KUKA KRL program: EPS_2_251806_MH06A_A_20260223023031.src

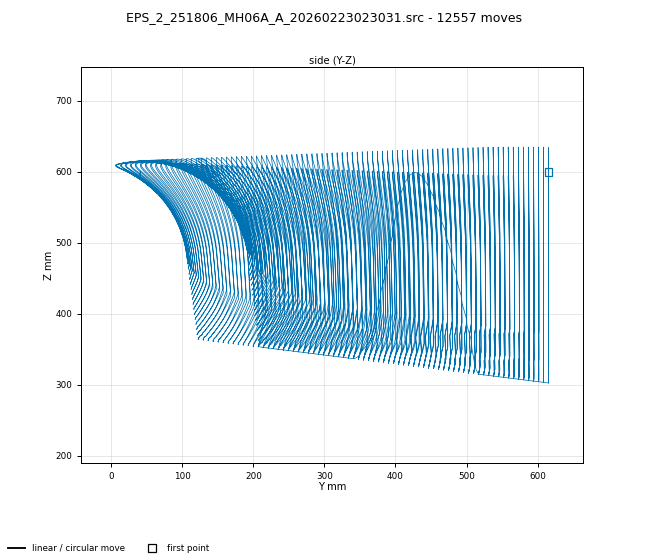
[picture p0: tool path of EPS_2_251806_MH06A_A_20260223023031.src, 12557 of 12559 moves have a stored position in this frame; points joined in program order, loops and branches not executed]
&ACCESS RVP
&REL 4
&COMMENT QRS 19112012
&PARAM EDITMASK = *
DEF PART()
EXT BAS (BAS_COMMAND :IN,REAL :IN )
INT I
BAS (#INITMOV,0 )

;KUKA QRS Post kuka4.cps  Date:22-06-2017 !

File_ID=3074

QRS_PRE_INIT()

;Init var - Until changes are made in qrs_pre_init
Outlet_Square_prg=0
Inlet_1_Square_prg=0
Inlet_2_Square_prg=0
Inlet_3_Square_prg=0
Inlet_4_Square_prg=0
Inlet_5_Square_prg=0

Outlet_1={X 0.000, Y 527.380, Z 509.000, B 0.000, E1 0.000 }
Inlet_1={X 0.000, Y 530.260, Z 469.000, B 0.000, E1 162.000 }
Outlet_1_type=251
Inlet_1_type=251
;QRS#1=Sidecore dimensions
;QRS#2=250-10" PVC SDR 35
;QRS#3=250-10" PVC SDR 35
;QRS#4=
;QRS#5=
;QRS#6=
;QRS#7=
;QRS#8=
;QRS#9=14M PSX
;QRS#10=14M PSX
;QRS#11=
;QRS#12=
;QRS#13=
;QRS#14=
;QRS#15=
;QRS#16=1220x127x914 3'
;QRS#17=EPS Height
;QRS#18=634,5
;QRS#19=*
;QRS#20= UPDATED VERSION 22-06-2017
;QRS#21=*
Outlet_Square=0100
Inlet_1_Square=0100
Inlet_2_Square=0
Inlet_3_Square=0
Inlet_4_Square=0
Inlet_5_Square=0
Mill_Square=1
Outlet_Square_Prg=205
Inlet_1_Square_prg=205

QRS_INIT()

$ADVANCE=5

; T1
PTP {E1 173.655,E2 173.655}
PTP {X 0,Y 615.421,A -85,B 0,C 180,E1 173.655,E2 173.655,E3 0,E4 0,E5 0,E6 0}
QRS_SPEED_INIT()
LIN {X 0,Y 615.421,Z 600,A -85,B 0,C 180,E1 173.655,E2 173.655,E3 0,E4 0,E5 0,E6 0} C_VEL
LIN {X 0,Y 615.421,Z 312.502,A -85,B 0,C 180,E1 173.655,E2 173.655} C_VEL
LIN {X 0,Y 615.421,Z 304.323,A -85,B 0,C 180,E1 173.655,E2 173.655} C_VEL
LIN {X 0,Y 615.418,Z 302.323,A -85,B 0,C 180,E1 173.469,E2 173.469} C_VEL
LIN {X 0,Y 615.458,Z 302.323,A -85,B 0,C 180,E1 170.801,E2 170.801} C_VEL
LIN {X 0,Y 615.445,Z 302.325,A -85,B 0,C 180,E1 168.139,E2 168.139} C_VEL
LIN {X 0,Y 615.434,Z 302.325,A -85,B 0,C 180,E1 166.083,E2 166.083} C_VEL
LIN {X 0,Y 615.411,Z 302.325,A -85,B 0,C 180,E1 163.589,E2 163.589} C_VEL
LIN {X 0,Y 615.423,Z 302.324,A -85,B 0,C 180,E1 161.352,E2 161.352} C_VEL
LIN {X 0,Y 615.489,Z 302.322,A -85,B 0,C 180,E1 158.568,E2 158.568} C_VEL
LIN {X 0,Y 615.423,Z 302.322,A -85,B 0,C 180,E1 155.726,E2 155.726} C_VEL
LIN {X 0,Y 615.484,Z 302.325,A -85,B 0,C 180,E1 152.953,E2 152.953} C_VEL
LIN {X 0,Y 615.446,Z 302.319,A -85,B 0,C 180,E1 150.21,E2 150.21} C_VEL
LIN {X 0,Y 615.435,Z 302.321,A -85,B 0,C 180,E1 147.675,E2 147.675} C_VEL
LIN {X 0,Y 615.476,Z 302.324,A -85,B 0,C 180,E1 145.185,E2 145.185} C_VEL
LIN {X 0,Y 615.492,Z 302.317,A -85,B 0,C 180,E1 142.759,E2 142.759} C_VEL
LIN {X 0,Y 615.452,Z 302.316,A -85,B 0,C 180,E1 140.247,E2 140.247} C_VEL
LIN {X 0,Y 615.453,Z 302.321,A -85,B 0,C 180,E1 137.645,E2 137.645} C_VEL
LIN {X 0,Y 615.489,Z 302.317,A -85,B 0,C 180,E1 134.932,E2 134.932} C_VEL
LIN {X 0,Y 615.456,Z 302.315,A -85,B 0,C 180,E1 132.354,E2 132.354} C_VEL
LIN {X 0,Y 615.46,Z 302.321,A -85,B 0,C 180,E1 129.751,E2 129.751} C_VEL
LIN {X 0,Y 615.455,Z 302.33,A -85,B 0,C 180,E1 128.039,E2 128.039} C_VEL
LIN {X 0,Y 615.471,Z 320.019,A -85,B 0,C 180,E1 125.415,E2 125.415} C_VEL
LIN {X 0,Y 615.484,Z 332.842,A -85,B 0,C 180,E1 123.534,E2 123.534} C_VEL
LIN {X 0,Y 615.493,Z 469.157,A -85,B 0,C 180,E1 121.905,E2 121.905} C_VEL
LIN {X 0,Y 615.496,Z 483.195,A -85,B 0,C 180,E1 121.609,E2 121.609} C_VEL
LIN {X 0,Y 615.493,Z 497.538,A -85,B 0,C 180,E1 121.162,E2 121.162} C_VEL
LIN {X 0,Y 615.494,Z 510.249,A -85,B 0,C 180,E1 120.633,E2 120.633} C_VEL
LIN {X 0,Y 615.49,Z 522.679,A -85,B 0,C 180,E1 119.978,E2 119.978} C_VEL
LIN {X 0,Y 615.497,Z 534.378,A -85,B 0,C 180,E1 119.217,E2 119.217} C_VEL
LIN {X 0,Y 615.498,Z 545.719,A -85,B 0,C 180,E1 118.318,E2 118.318} C_VEL
LIN {X 0,Y 615.496,Z 555.694,A -85,B 0,C 180,E1 117.36,E2 117.36} C_VEL
LIN {X 0,Y 615.495,Z 565.103,A -85,B 0,C 180,E1 116.26,E2 116.26} C_VEL
LIN {X 0,Y 615.495,Z 572.038,A -85,B 0,C 180,E1 115.281,E2 115.281} C_VEL
LIN {X 0,Y 615.495,Z 579.304,A -85,B 0,C 180,E1 114.011,E2 114.011} C_VEL
LIN {X 0,Y 615.493,Z 584.548,A -85,B 0,C 180,E1 112.843,E2 112.843} C_VEL
LIN {X 0,Y 615.498,Z 588.224,A -85,B 0,C 180,E1 111.783,E2 111.783} C_VEL
LIN {X 0,Y 615.493,Z 591.282,A -85,B 0,C 180,E1 110.559,E2 110.559} C_VEL
LIN {X 0,Y 615.491,Z 593.141,A -85,B 0,C 180,E1 109.337,E2 109.337} C_VEL
LIN {X 0,Y 615.498,Z 593.888,A -85,B 0,C 180,E1 107.956,E2 107.956} C_VEL
LIN {X 0,Y 615.489,Z 593.157,A -85,B 0,C 180,E1 106.586,E2 106.586} C_VEL
LIN {X 0,Y 615.493,Z 591.009,A -85,B 0,C 180,E1 105.225,E2 105.225} C_VEL
LIN {X 0,Y 615.499,Z 587.409,A -85,B 0,C 180,E1 103.873,E2 103.873} C_VEL
LIN {X 0,Y 615.491,Z 582.289,A -85,B 0,C 180,E1 102.529,E2 102.529} C_VEL
LIN {X 0,Y 615.496,Z 577.325,A -85,B 0,C 180,E1 101.526,E2 101.526} C_VEL
LIN {X 0,Y 615.496,Z 570.217,A -85,B 0,C 180,E1 100.36,E2 100.36} C_VEL
LIN {X 0,Y 615.496,Z 561.453,A -85,B 0,C 180,E1 99.198,E2 99.198} C_VEL
LIN {X 0,Y 615.497,Z 552.328,A -85,B 0,C 180,E1 98.205,E2 98.205} C_VEL
LIN {X 0,Y 615.496,Z 542.286,A -85,B 0,C 180,E1 97.297,E2 97.297} C_VEL
LIN {X 0,Y 615.5,Z 531.281,A -85,B 0,C 180,E1 96.474,E2 96.474} C_VEL
LIN {X 0,Y 615.489,Z 519.214,A -85,B 0,C 180,E1 95.733,E2 95.733} C_VEL
LIN {X 0,Y 615.495,Z 507.699,A -85,B 0,C 180,E1 95.158,E2 95.158} C_VEL
LIN {X 0,Y 615.496,Z 494.032,A -85,B 0,C 180,E1 94.625,E2 94.625} C_VEL
LIN {X 0,Y 615.492,Z 481.391,A -85,B 0,C 180,E1 94.256,E2 94.256} C_VEL
LIN {X 0,Y 615.492,Z 468.115,A -85,B 0,C 180,E1 93.989,E2 93.989} C_VEL
LIN {X 0,Y 615.476,Z 332.816,A -85,B 0,C 180,E1 92.372,E2 92.372} C_VEL
LIN {X 0,Y 615.478,Z 314.441,A -85,B 0,C 180,E1 89.672,E2 89.672} C_VEL
LIN {X 0,Y 615.448,Z 302.319,A -85,B 0,C 180,E1 87.852,E2 87.852} C_VEL
LIN {X 0,Y 615.458,Z 302.315,A -85,B 0,C 180,E1 85.415,E2 85.415} C_VEL
LIN {X 0,Y 615.494,Z 302.32,A -85,B 0,C 180,E1 82.784,E2 82.784} C_VEL
LIN {X 0,Y 615.448,Z 302.321,A -85,B 0,C 180,E1 80.137,E2 80.137} C_VEL
LIN {X 0,Y 615.445,Z 302.321,A -85,B 0,C 180,E1 78.138,E2 78.138} C_VEL
LIN {X 0,Y 615.441,Z 302.321,A -85,B 0,C 180,E1 76.084,E2 76.084} C_VEL
LIN {X 0,Y 615.447,Z 302.317,A -85,B 0,C 180,E1 73.581,E2 73.581} C_VEL
LIN {X 0,Y 615.477,Z 302.324,A -85,B 0,C 180,E1 70.661,E2 70.661} C_VEL
LIN {X 0,Y 615.458,Z 302.325,A -85,B 0,C 180,E1 68.567,E2 68.567} C_VEL
LIN {X 0,Y 615.429,Z 302.321,A -85,B 0,C 180,E1 66.003,E2 66.003} C_VEL
LIN {X 0,Y 615.448,Z 302.32,A -85,B 0,C 180,E1 63.554,E2 63.554} C_VEL
LIN {X 0,Y 615.448,Z 302.324,A -85,B 0,C 180,E1 60.591,E2 60.591} C_VEL
LIN {X 0,Y 615.426,Z 302.323,A -85,B 0,C 180,E1 58.311,E2 58.311} C_VEL
LIN {X 0,Y 615.422,Z 302.323,A -85,B 0,C 180,E1 55.974,E2 55.974} C_VEL
LIN {X 0,Y 615.449,Z 302.322,A -85,B 0,C 180,E1 53.572,E2 53.572} C_VEL
LIN {X 0,Y 615.467,Z 302.325,A -85,B 0,C 180,E1 50.94,E2 50.94} C_VEL
LIN {X 0,Y 615.421,Z 302.325,A -85,B 0,C 180,E1 48.52,E2 48.52} C_VEL
LIN {X 0,Y 615.424,Z 302.325,A -85,B 0,C 180,E1 45.844,E2 45.844} C_VEL
LIN {X 0,Y 615.466,Z 302.324,A -85,B 0,C 180,E1 43.045,E2 43.045} C_VEL
LIN {X 0,Y 615.422,Z 302.324,A -85,B 0,C 180,E1 40.611,E2 40.611} C_VEL
LIN {X 0,Y 615.426,Z 302.324,A -85,B 0,C 180,E1 38.004,E2 38.004} C_VEL
LIN {X 0,Y 615.469,Z 302.325,A -85,B 0,C 180,E1 35.617,E2 35.617} C_VEL
LIN {X 0,Y 615.483,Z 302.321,A -85,B 0,C 180,E1 33.236,E2 33.236} C_VEL
LIN {X 0,Y 615.447,Z 302.32,A -85,B 0,C 180,E1 30.922,E2 30.922} C_VEL
LIN {X 0,Y 615.426,Z 302.322,A -85,B 0,C 180,E1 28.439,E2 28.439} C_VEL
LIN {X 0,Y 615.476,Z 302.325,A -85,B 0,C 180,E1 25.716,E2 25.716} C_VEL
LIN {X 0,Y 615.438,Z 302.32,A -85,B 0,C 180,E1 22.846,E2 22.846} C_VEL
LIN {X 0,Y 615.433,Z 302.32,A -85,B 0,C 180,E1 20.543,E2 20.543} C_VEL
LIN {X 0,Y 615.467,Z 302.324,A -85,B 0,C 180,E1 17.957,E2 17.957} C_VEL
LIN {X 0,Y 615.475,Z 302.315,A -85,B 0,C 180,E1 15.226,E2 15.226} C_VEL
LIN {X 0,Y 615.44,Z 302.32,A -85,B 0,C 180,E1 12.531,E2 12.531} C_VEL
LIN {X 0,Y 615.497,Z 302.325,A -85,B 0,C 180,E1 9.862,E2 9.862} C_VEL
LIN {X 0,Y 615.47,Z 302.314,A -85,B 0,C 180,E1 7.216,E2 7.216} C_VEL
LIN {X 0,Y 615.473,Z 302.313,A -85,B 0,C 180,E1 5.241,E2 5.241} C_VEL
LIN {X 0,Y 615.447,Z 302.319,A -85,B 0,C 180,E1 2.618,E2 2.618} C_VEL
LIN {X 0,Y 615.487,Z 302.328,A -85,B 0,C 180,E1 0,E2 0} C_VEL
LIN {X 0,Y 615.484,Z 302.31,A -85,B 0,C 180,E1 -2.618,E2 -2.618} C_VEL
LIN {X 0,Y 615.454,Z 302.318,A -85,B 0,C 180,E1 -5.242,E2 -5.242} C_VEL
LIN {X 0,Y 615.487,Z 302.328,A -85,B 0,C 180,E1 -7.876,E2 -7.876} C_VEL
LIN {X 0,Y 615.49,Z 302.309,A -85,B 0,C 180,E1 -10.527,E2 -10.527} C_VEL
LIN {X 0,Y 615.46,Z 302.318,A -85,B 0,C 180,E1 -13.202,E2 -13.202} C_VEL
LIN {X 0,Y 615.491,Z 302.321,A -85,B 0,C 180,E1 -15.905,E2 -15.905} C_VEL
LIN {X 0,Y 615.477,Z 302.31,A -85,B 0,C 180,E1 -18.647,E2 -18.647} C_VEL
LIN {X 0,Y 615.481,Z 302.322,A -85,B 0,C 180,E1 -21.432,E2 -21.432} C_VEL
LIN {X 0,Y 615.491,Z 302.309,A -85,B 0,C 180,E1 -24.272,E2 -24.272} C_VEL
LIN {X 0,Y 615.469,Z 302.317,A -85,B 0,C 180,E1 -27.041,E2 -27.041} C_VEL
LIN {X 0,Y 615.482,Z 302.319,A -85,B 0,C 180,E1 -29.793,E2 -29.793} C_VEL
LIN {X 0,Y 615.488,Z 302.307,A -85,B 0,C 180,E1 -32.458,E2 -32.458} C_VEL
LIN {X 0,Y 615.473,Z 302.314,A -85,B 0,C 180,E1 -34.816,E2 -34.816} C_VEL
LIN {X 0,Y 615.484,Z 302.324,A -85,B 0,C 180,E1 -37.243,E2 -37.243} C_VEL
LIN {X 0,Y 615.487,Z 302.309,A -85,B 0,C 180,E1 -40.089,E2 -40.089} C_VEL
LIN {X 0,Y 615.493,Z 302.306,A -85,B 0,C 180,E1 -42.353,E2 -42.353} C_VEL
LIN {X 0,Y 615.48,Z 302.323,A -85,B 0,C 180,E1 -45.069,E2 -45.069} C_VEL
LIN {X 0,Y 615.479,Z 302.311,A -85,B 0,C 180,E1 -47.921,E2 -47.921} C_VEL
LIN {X 0,Y 615.494,Z 302.306,A -85,B 0,C 180,E1 -50.25,E2 -50.25} C_VEL
LIN {X 0,Y 615.485,Z 302.327,A -85,B 0,C 180,E1 -53.064,E2 -53.064} C_VEL
LIN {X 0,Y 615.481,Z 302.321,A -85,B 0,C 180,E1 -55.3,E2 -55.3} C_VEL
LIN {X 0,Y 615.468,Z 302.314,A -85,B 0,C 180,E1 -57.672,E2 -57.672} C_VEL
LIN {X 0,Y 615.497,Z 302.306,A -85,B 0,C 180,E1 -60.204,E2 -60.204} C_VEL
LIN {X 0,Y 615.498,Z 302.325,A -85,B 0,C 180,E1 -62.953,E2 -62.953} C_VEL
LIN {X 0,Y 615.469,Z 302.312,A -85,B 0,C 180,E1 -65.727,E2 -65.727} C_VEL
LIN {X 0,Y 615.483,Z 302.338,A -85,B 0,C 180,E1 -66.106,E2 -66.106} C_VEL
LIN {X 0,Y 615.484,Z 325.342,A -85,B 0,C 180,E1 -68.919,E2 -68.919} C_VEL
LIN {X 0,Y 615.5,Z 348.671,A -85,B 0,C 180,E1 -71.719,E2 -71.719} C_VEL
LIN {X 0,Y 615.483,Z 371.267,A -85,B 0,C 180,E1 -74.392,E2 -74.392} C_VEL
LIN {X 0,Y 615.498,Z 509.937,A -85,B 0,C 180,E1 -76.064,E2 -76.064} C_VEL
LIN {X 0,Y 615.495,Z 524.359,A -85,B 0,C 180,E1 -76.378,E2 -76.378} C_VEL
LIN {X 0,Y 615.489,Z 537.675,A -85,B 0,C 180,E1 -76.798,E2 -76.798} C_VEL
LIN {X 0,Y 615.498,Z 551.571,A -85,B 0,C 180,E1 -77.386,E2 -77.386} C_VEL
LIN {X 0,Y 615.495,Z 563.999,A -85,B 0,C 180,E1 -78.055,E2 -78.055} C_VEL
LIN {X 0,Y 615.499,Z 575.333,A -85,B 0,C 180,E1 -78.807,E2 -78.807} C_VEL
LIN {X 0,Y 615.498,Z 585.742,A -85,B 0,C 180,E1 -79.639,E2 -79.639} C_VEL
LIN {X 0,Y 615.496,Z 596.083,A -85,B 0,C 180,E1 -80.635,E2 -80.635} C_VEL
LIN {X 0,Y 615.497,Z 604.598,A -85,B 0,C 180,E1 -81.628,E2 -81.628} C_VEL
LIN {X 0,Y 615.496,Z 612.723,A -85,B 0,C 180,E1 -82.784,E2 -82.784} C_VEL
LIN {X 0,Y 615.496,Z 618.427,A -85,B 0,C 180,E1 -83.772,E2 -83.772} C_VEL
LIN {X 0,Y 615.495,Z 623.078,A -85,B 0,C 180,E1 -84.758,E2 -84.758} C_VEL
LIN {X 0,Y 615.494,Z 627.9,A -85,B 0,C 180,E1 -86.071,E2 -86.071} C_VEL
LIN {X 0,Y 615.496,Z 631.251,A -85,B 0,C 180,E1 -87.382,E2 -87.382} C_VEL
LIN {X 0,Y 615.489,Z 633.228,A -85,B 0,C 180,E1 -88.691,E2 -88.691} C_VEL
LIN {X 0,Y 615.493,Z 633.889,A -85,B 0,C 180,E1 -89.999,E2 -89.999} C_VEL
LIN {X 0,Y 615.489,Z 633.229,A -85,B 0,C 180,E1 -91.308,E2 -91.308} C_VEL
LIN {X 0,Y 615.496,Z 631.253,A -85,B 0,C 180,E1 -92.617,E2 -92.617} C_VEL
LIN {X 0,Y 615.494,Z 627.904,A -85,B 0,C 180,E1 -93.928,E2 -93.928} C_VEL
LIN {X 0,Y 615.495,Z 623.083,A -85,B 0,C 180,E1 -95.24,E2 -95.24} C_VEL
LIN {X 0,Y 615.496,Z 616.632,A -85,B 0,C 180,E1 -96.556,E2 -96.556} C_VEL
LIN {X 0,Y 615.497,Z 609.445,A -85,B 0,C 180,E1 -97.71,E2 -97.71} C_VEL
LIN {X 0,Y 615.497,Z 601.908,A -85,B 0,C 180,E1 -98.701,E2 -98.701} C_VEL
LIN {X 0,Y 615.495,Z 592.859,A -85,B 0,C 180,E1 -99.695,E2 -99.695} C_VEL
LIN {X 0,Y 615.497,Z 582.763,A -85,B 0,C 180,E1 -100.618,E2 -100.618} C_VEL
LIN {X 0,Y 615.498,Z 571.867,A -85,B 0,C 180,E1 -101.442,E2 -101.442} C_VEL
LIN {X 0,Y 615.489,Z 559.718,A -85,B 0,C 180,E1 -102.195,E2 -102.195} C_VEL
LIN {X 0,Y 615.498,Z 546.106,A -85,B 0,C 180,E1 -102.865,E2 -102.865} C_VEL
LIN {X 0,Y 615.49,Z 532.855,A -85,B 0,C 180,E1 -103.368,E2 -103.368} C_VEL
LIN {X 0,Y 615.494,Z 519.315,A -85,B 0,C 180,E1 -103.747,E2 -103.747} C_VEL
LIN {X 0,Y 615.493,Z 504.752,A -85,B 0,C 180,E1 -104.013,E2 -104.013} C_VEL
LIN {X 0,Y 615.483,Z 371.277,A -85,B 0,C 180,E1 -105.607,E2 -105.607} C_VEL
LIN {X 0,Y 615.49,Z 347.317,A -85,B 0,C 180,E1 -108.442,E2 -108.442} C_VEL
LIN {X 0,Y 615.486,Z 325.352,A -85,B 0,C 180,E1 -111.08,E2 -111.08} C_VEL
LIN {X 0,Y 615.484,Z 302.309,A -85,B 0,C 180,E1 -113.908,E2 -113.908} C_VEL
LIN {X 0,Y 615.466,Z 302.316,A -85,B 0,C 180,E1 -116.444,E2 -116.444} C_VEL
LIN {X 0,Y 615.474,Z 302.319,A -85,B 0,C 180,E1 -118.658,E2 -118.658} C_VEL
LIN {X 0,Y 615.485,Z 302.324,A -85,B 0,C 180,E1 -121.085,E2 -121.085} C_VEL
LIN {X 0,Y 615.482,Z 302.309,A -85,B 0,C 180,E1 -124.021,E2 -124.021} C_VEL
LIN {X 0,Y 615.476,Z 302.317,A -85,B 0,C 180,E1 -126.424,E2 -126.424} C_VEL
LIN {X 0,Y 615.482,Z 302.32,A -85,B 0,C 180,E1 -129.061,E2 -129.061} C_VEL
LIN {X 0,Y 615.48,Z 302.311,A -85,B 0,C 180,E1 -131.473,E2 -131.473} C_VEL
LIN {X 0,Y 615.481,Z 302.314,A -85,B 0,C 180,E1 -134.149,E2 -134.149} C_VEL
LIN {X 0,Y 615.477,Z 302.319,A -85,B 0,C 180,E1 -136.952,E2 -136.952} C_VEL
LIN {X 0,Y 615.475,Z 302.311,A -85,B 0,C 180,E1 -139.392,E2 -139.392} C_VEL
LIN {X 0,Y 615.487,Z 302.312,A -85,B 0,C 180,E1 -141.987,E2 -141.987} C_VEL
LIN {X 0,Y 615.495,Z 302.323,A -85,B 0,C 180,E1 -144.384,E2 -144.384} C_VEL
LIN {X 0,Y 615.471,Z 302.32,A -85,B 0,C 180,E1 -146.763,E2 -146.763} C_VEL
LIN {X 0,Y 615.462,Z 302.315,A -85,B 0,C 180,E1 -149.079,E2 -149.079} C_VEL
LIN {X 0,Y 615.488,Z 302.309,A -85,B 0,C 180,E1 -151.548,E2 -151.548} C_VEL
LIN {X 0,Y 615.481,Z 302.323,A -85,B 0,C 180,E1 -154.43,E2 -154.43} C_VEL
LIN {X 0,Y 615.459,Z 302.314,A -85,B 0,C 180,E1 -157.154,E2 -157.154} C_VEL
LIN {X 0,Y 615.493,Z 302.32,A -85,B 0,C 180,E1 -159.967,E2 -159.967} C_VEL
LIN {X 0,Y 615.447,Z 302.319,A -85,B 0,C 180,E1 -162.728,E2 -162.728} C_VEL
LIN {X 0,Y 615.484,Z 302.312,A -85,B 0,C 180,E1 -165.451,E2 -165.451} C_VEL
LIN {X 0,Y 615.479,Z 302.324,A -85,B 0,C 180,E1 -168.139,E2 -168.139} C_VEL
LIN {X 0,Y 615.44,Z 302.319,A -85,B 0,C 180,E1 -170.8,E2 -170.8} C_VEL
LIN {X 0,Y 615.487,Z 302.315,A -85,B 0,C 180,E1 -173.443,E2 -173.443} C_VEL
LIN {X 0,Y 615.465,Z 302.324,A -85,B 0,C 180,E1 -176.071,E2 -176.071} C_VEL
LIN {X 0,Y 615.429,Z 302.321,A -85,B 0,C 180,E1 -178.691,E2 -178.691} C_VEL
LIN {X 0,Y 615.473,Z 302.319,A -85,B 0,C 180,E1 -181.308,E2 -181.308} C_VEL
LIN {X 0,Y 615.46,Z 302.324,A -85,B 0,C 180,E1 -183.928,E2 -183.928} C_VEL
LIN {X 0,Y 615.418,Z 302.323,A -85,B 0,C 180,E1 -186.531,E2 -186.531} C_VEL
LIN {X 0,Y 614.771,Z 302.471,A -85,B 0,C 180,E1 -187.077,E2 -187.077} C_VEL
LIN {X 0,Y 611.962,Z 302.879,A -85,B 0,C 180,E1 -187.963,E2 -187.963} C_VEL
LIN {X 0,Y 609.571,Z 303.192,A -85,B 0,C 180,E1 -188.676,E2 -188.676} C_VEL
LIN {X 0,Y 608.527,Z 303.311,A -85,B 0,C 180,E1 -189.225,E2 -189.225} C_VEL
LIN {X 0,Y 608.433,Z 303.32,A -85,B 0,C 180,E1 -189.412,E2 -189.412} C_VEL
LIN {X 0,Y 608.418,Z 303.319,A -85,B 0,C 180,E1 -192,E2 -192} C_VEL
LIN {X 0,Y 608.406,Z 303.32,A -85,B 0,C 180,E1 -194.039,E2 -194.039} C_VEL
LIN {X 0,Y 608.384,Z 303.321,A -85,B 0,C 180,E1 -196.506,E2 -196.506} C_VEL
LIN {X 0,Y 608.425,Z 303.319,A -85,B 0,C 180,E1 -198.87,E2 -198.87} C_VEL
LIN {X 0,Y 608.447,Z 303.317,A -85,B 0,C 180,E1 -201.692,E2 -201.692} C_VEL
LIN {X 0,Y 608.416,Z 303.319,A -85,B 0,C 180,E1 -204.572,E2 -204.572} C_VEL
LIN {X 0,Y 608.477,Z 303.319,A -85,B 0,C 180,E1 -207.209,E2 -207.209} C_VEL
LIN {X 0,Y 608.409,Z 303.318,A -85,B 0,C 180,E1 -209.964,E2 -209.964} C_VEL
LIN {X 0,Y 608.422,Z 303.319,A -85,B 0,C 180,E1 -212.518,E2 -212.518} C_VEL
LIN {X 0,Y 608.425,Z 303.321,A -85,B 0,C 180,E1 -215.278,E2 -215.278} C_VEL
LIN {X 0,Y 608.442,Z 303.314,A -85,B 0,C 180,E1 -217.748,E2 -217.748} C_VEL
LIN {X 0,Y 608.422,Z 303.318,A -85,B 0,C 180,E1 -220.327,E2 -220.327} C_VEL
LIN {X 0,Y 608.455,Z 303.32,A -85,B 0,C 180,E1 -222.959,E2 -222.959} C_VEL
LIN {X 0,Y 608.425,Z 303.316,A -85,B 0,C 180,E1 -225.739,E2 -225.739} C_VEL
LIN {X 0,Y 608.43,Z 303.316,A -85,B 0,C 180,E1 -227.937,E2 -227.937} C_VEL
LIN {X 0,Y 608.471,Z 303.321,A -85,B 0,C 180,E1 -230.702,E2 -230.702} C_VEL
LIN {X 0,Y 608.45,Z 303.347,A -85,B 0,C 180,E1 -231.87,E2 -231.87} C_VEL
LIN {X 0,Y 608.5,Z 319.687,A -85,B 0,C 180,E1 -234.321,E2 -234.321} C_VEL
LIN {X 0,Y 608.532,Z 333.181,A -85,B 0,C 180,E1 -236.289,E2 -236.289} C_VEL
LIN {X 0,Y 608.603,Z 469.47,A -85,B 0,C 180,E1 -237.939,E2 -237.939} C_VEL
LIN {X 0,Y 608.596,Z 483.994,A -85,B 0,C 180,E1 -238.255,E2 -238.255} C_VEL
LIN {X 0,Y 608.56,Z 497.685,A -85,B 0,C 180,E1 -238.69,E2 -238.69} C_VEL
LIN {X 0,Y 608.538,Z 511.282,A -85,B 0,C 180,E1 -239.268,E2 -239.268} C_VEL
LIN {X 0,Y 608.529,Z 523.689,A -85,B 0,C 180,E1 -239.938,E2 -239.938} C_VEL
LIN {X 0,Y 608.518,Z 535.16,A -85,B 0,C 180,E1 -240.699,E2 -240.699} C_VEL
LIN {X 0,Y 608.503,Z 546.875,A -85,B 0,C 180,E1 -241.646,E2 -241.646} C_VEL
LIN {X 0,Y 608.476,Z 557.274,A -85,B 0,C 180,E1 -242.674,E2 -242.674} C_VEL
LIN {X 0,Y 608.465,Z 566.452,A -85,B 0,C 180,E1 -243.782,E2 -243.782} C_VEL
LIN {X 0,Y 608.454,Z 573.946,A -85,B 0,C 180,E1 -244.883,E2 -244.883} C_VEL
LIN {X 0,Y 608.444,Z 580.901,A -85,B 0,C 180,E1 -246.155,E2 -246.155} C_VEL
LIN {X 0,Y 608.422,Z 585.559,A -85,B 0,C 180,E1 -247.235,E2 -247.235} C_VEL
LIN {X 0,Y 608.427,Z 589.176,A -85,B 0,C 180,E1 -248.308,E2 -248.308} C_VEL
LIN {X 0,Y 608.435,Z 592.445,A -85,B 0,C 180,E1 -249.726,E2 -249.726} C_VEL
LIN {X 0,Y 608.424,Z 594.154,A -85,B 0,C 180,E1 -251.13,E2 -251.13} C_VEL
LIN {X 0,Y 608.415,Z 594.394,A -85,B 0,C 180,E1 -252.523,E2 -252.523} C_VEL
LIN {X 0,Y 608.431,Z 593.195,A -85,B 0,C 180,E1 -253.906,E2 -253.906} C_VEL
LIN {X 0,Y 608.42,Z 590.521,A -85,B 0,C 180,E1 -255.279,E2 -255.279} C_VEL
LIN {X 0,Y 608.441,Z 586.343,A -85,B 0,C 180,E1 -256.644,E2 -256.644} C_VEL
LIN {X 0,Y 608.444,Z 580.582,A -85,B 0,C 180,E1 -258.001,E2 -258.001} C_VEL
LIN {X 0,Y 608.435,Z 574.844,A -85,B 0,C 180,E1 -259.059,E2 -259.059} C_VEL
LIN {X 0,Y 608.45,Z 567.318,A -85,B 0,C 180,E1 -260.191,E2 -260.191} C_VEL
LIN {X 0,Y 608.475,Z 559.21,A -85,B 0,C 180,E1 -261.198,E2 -261.198} C_VEL
LIN {X 0,Y 608.492,Z 549.496,A -85,B 0,C 180,E1 -262.201,E2 -262.201} C_VEL
LIN {X 0,Y 608.511,Z 538.671,A -85,B 0,C 180,E1 -263.127,E2 -263.127} C_VEL
LIN {X 0,Y 608.532,Z 526.982,A -85,B 0,C 180,E1 -263.951,E2 -263.951} C_VEL
LIN {X 0,Y 608.532,Z 513.82,A -85,B 0,C 180,E1 -264.699,E2 -264.699} C_VEL
LIN {X 0,Y 608.575,Z 500.825,A -85,B 0,C 180,E1 -265.281,E2 -265.281} C_VEL
LIN {X 0,Y 608.589,Z 486.737,A -85,B 0,C 180,E1 -265.758,E2 -265.758} C_VEL
LIN {X 0,Y 608.604,Z 472.745,A -85,B 0,C 180,E1 -266.09,E2 -266.09} C_VEL
LIN {X 0,Y 608.618,Z 453.41,A -85,B 0,C 180,E1 -266.359,E2 -266.359} C_VEL
LIN {X 0,Y 608.493,Z 332.936,A -85,B 0,C 180,E1 -267.808,E2 -267.808} C_VEL
LIN {X 0,Y 608.514,Z 313.697,A -85,B 0,C 180,E1 -270.662,E2 -270.662} C_VEL
LIN {X 0,Y 608.434,Z 303.317,A -85,B 0,C 180,E1 -272.235,E2 -272.235} C_VEL
LIN {X 0,Y 608.43,Z 303.316,A -85,B 0,C 180,E1 -274.638,E2 -274.638} C_VEL
LIN {X 0,Y 608.484,Z 303.318,A -85,B 0,C 180,E1 -277.3,E2 -277.3} C_VEL
LIN {X 0,Y 608.421,Z 303.318,A -85,B 0,C 180,E1 -279.978,E2 -279.978} C_VEL
LIN {X 0,Y 608.428,Z 303.316,A -85,B 0,C 180,E1 -282.001,E2 -282.001} C_VEL
LIN {X 0,Y 608.417,Z 303.317,A -85,B 0,C 180,E1 -284.039,E2 -284.039} C_VEL
LIN {X 0,Y 608.445,Z 303.314,A -85,B 0,C 180,E1 -286.523,E2 -286.523} C_VEL
LIN {X 0,Y 608.43,Z 303.319,A -85,B 0,C 180,E1 -289.572,E2 -289.572} C_VEL
LIN {X 0,Y 608.431,Z 303.316,A -85,B 0,C 180,E1 -292.407,E2 -292.407} C_VEL
LIN {X 0,Y 608.429,Z 303.322,A -85,B 0,C 180,E1 -295.302,E2 -295.302} C_VEL
LIN {X 0,Y 608.423,Z 303.319,A -85,B 0,C 180,E1 -297.52,E2 -297.52} C_VEL
LIN {X 0,Y 608.395,Z 303.32,A -85,B 0,C 180,E1 -299.96,E2 -299.96} C_VEL
LIN {X 0,Y 608.432,Z 303.318,A -85,B 0,C 180,E1 -302.519,E2 -302.519} C_VEL
LIN {X 0,Y 608.414,Z 303.322,A -85,B 0,C 180,E1 -305.28,E2 -305.28} C_VEL
LIN {X 0,Y 608.396,Z 303.319,A -85,B 0,C 180,E1 -307.752,E2 -307.752} C_VEL
LIN {X 0,Y 608.432,Z 303.318,A -85,B 0,C 180,E1 -310.327,E2 -310.327} C_VEL
LIN {X 0,Y 608.428,Z 303.318,A -85,B 0,C 180,E1 -313.305,E2 -313.305} C_VEL
LIN {X 0,Y 608.418,Z 303.318,A -85,B 0,C 180,E1 -316.126,E2 -316.126} C_VEL
LIN {X 0,Y 608.439,Z 303.322,A -85,B 0,C 180,E1 -318.822,E2 -318.822} C_VEL
LIN {X 0,Y 608.396,Z 303.32,A -85,B 0,C 180,E1 -321.407,E2 -321.407} C_VEL
LIN {X 0,Y 608.424,Z 303.317,A -85,B 0,C 180,E1 -323.907,E2 -323.907} C_VEL
LIN {X 0,Y 608.443,Z 303.32,A -85,B 0,C 180,E1 -326.328,E2 -326.328} C_VEL
LIN {X 0,Y 608.44,Z 303.321,A -85,B 0,C 180,E1 -328.734,E2 -328.734} C_VEL
LIN {X 0,Y 608.424,Z 303.316,A -85,B 0,C 180,E1 -331.389,E2 -331.389} C_VEL
LIN {X 0,Y 608.416,Z 303.32,A -85,B 0,C 180,E1 -333.963,E2 -333.963} C_VEL
LIN {X 0,Y 608.426,Z 303.318,A -85,B 0,C 180,E1 -336.875,E2 -336.875} C_VEL
LIN {X 0,Y 608.427,Z 303.316,A -85,B 0,C 180,E1 -339.332,E2 -339.332} C_VEL
LIN {X 0,Y 608.419,Z 303.32,A -85,B 0,C 180,E1 -341.827,E2 -341.827} C_VEL
LIN {X 0,Y 608.46,Z 303.316,A -85,B 0,C 180,E1 -344.594,E2 -344.594} C_VEL
LIN {X 0,Y 608.415,Z 303.317,A -85,B 0,C 180,E1 -347.322,E2 -347.322} C_VEL
LIN {X 0,Y 608.457,Z 303.32,A -85,B 0,C 180,E1 -350.023,E2 -350.023} C_VEL
LIN {X 0,Y 608.439,Z 303.316,A -85,B 0,C 180,E1 -352.701,E2 -352.701} C_VEL
LIN {X 0,Y 608.455,Z 303.314,A -85,B 0,C 180,E1 -354.698,E2 -354.698} C_VEL
LIN {X 0,Y 608.443,Z 303.315,A -85,B 0,C 180,E1 -357.352,E2 -357.352} C_VEL
LIN {X 0,Y 608.477,Z 303.32,A -85,B 0,C 180,E1 -360,E2 -360} C_VEL
LIN {X 0,Y 608.474,Z 303.311,A -85,B 0,C 180,E1 -362.648,E2 -362.648} C_VEL
LIN {X 0,Y 608.439,Z 303.316,A -85,B 0,C 180,E1 -365.302,E2 -365.302} C_VEL
LIN {X 0,Y 608.478,Z 303.318,A -85,B 0,C 180,E1 -367.967,E2 -367.967} C_VEL
LIN {X 0,Y 608.458,Z 303.312,A -85,B 0,C 180,E1 -370.949,E2 -370.949} C_VEL
LIN {X 0,Y 608.447,Z 303.317,A -85,B 0,C 180,E1 -373.357,E2 -373.357} C_VEL
LIN {X 0,Y 608.465,Z 303.315,A -85,B 0,C 180,E1 -376.094,E2 -376.094} C_VEL
LIN {X 0,Y 608.45,Z 303.313,A -85,B 0,C 180,E1 -378.87,E2 -378.87} C_VEL
LIN {X 0,Y 608.465,Z 303.321,A -85,B 0,C 180,E1 -381.692,E2 -381.692} C_VEL
LIN {X 0,Y 608.449,Z 303.313,A -85,B 0,C 180,E1 -384.571,E2 -384.571} C_VEL
LIN {X 0,Y 608.469,Z 303.315,A -85,B 0,C 180,E1 -387.205,E2 -387.205} C_VEL
LIN {X 0,Y 608.466,Z 303.314,A -85,B 0,C 180,E1 -389.971,E2 -389.971} C_VEL
LIN {X 0,Y 608.458,Z 303.314,A -85,B 0,C 180,E1 -392.88,E2 -392.88} C_VEL
LIN {X 0,Y 608.439,Z 303.323,A -85,B 0,C 180,E1 -395.278,E2 -395.278} C_VEL
LIN {X 0,Y 608.468,Z 303.315,A -85,B 0,C 180,E1 -397.747,E2 -397.747} C_VEL
LIN {X 0,Y 608.449,Z 303.313,A -85,B 0,C 180,E1 -400.328,E2 -400.328} C_VEL
LIN {X 0,Y 608.483,Z 303.319,A -85,B 0,C 180,E1 -403.31,E2 -403.31} C_VEL
LIN {X 0,Y 608.468,Z 303.311,A -85,B 0,C 180,E1 -406.13,E2 -406.13} C_VEL
LIN {X 0,Y 608.453,Z 303.317,A -85,B 0,C 180,E1 -408.823,E2 -408.823} C_VEL
LIN {X 0,Y 608.471,Z 303.316,A -85,B 0,C 180,E1 -411.412,E2 -411.412} C_VEL
LIN {X 0,Y 608.449,Z 303.313,A -85,B 0,C 180,E1 -413.954,E2 -413.954} C_VEL
LIN {X 0,Y 608.451,Z 303.313,A -85,B 0,C 180,E1 -416.328,E2 -416.328} C_VEL
LIN {X 0,Y 608.45,Z 303.319,A -85,B 0,C 180,E1 -418.732,E2 -418.732} C_VEL
LIN {X 0,Y 608.46,Z 303.315,A -85,B 0,C 180,E1 -421.383,E2 -421.383} C_VEL
LIN {X 0,Y 608.44,Z 303.314,A -85,B 0,C 180,E1 -423.964,E2 -423.964} C_VEL
LIN {X 0,Y 608.484,Z 303.496,A -85,B 0,C 180,E1 -425.959,E2 -425.959} C_VEL
LIN {X 0,Y 608.598,Z 318.101,A -85,B 0,C 180,E1 -427.778,E2 -427.778} C_VEL
LIN {X 0,Y 608.579,Z 339.823,A -85,B 0,C 180,E1 -430.433,E2 -430.433} C_VEL
LIN {X 0,Y 608.526,Z 362.995,A -85,B 0,C 180,E1 -433.218,E2 -433.218} C_VEL
LIN {X 0,Y 608.51,Z 371.412,A -85,B 0,C 180,E1 -434.219,E2 -434.219} C_VEL
LIN {X 0,Y 608.617,Z 509.424,A -85,B 0,C 180,E1 -435.894,E2 -435.894} C_VEL
LIN {X 0,Y 608.594,Z 523.606,A -85,B 0,C 180,E1 -436.199,E2 -436.199} C_VEL
LIN {X 0,Y 608.579,Z 537.697,A -85,B 0,C 180,E1 -436.646,E2 -436.646} C_VEL
LIN {X 0,Y 608.565,Z 549.872,A -85,B 0,C 180,E1 -437.155,E2 -437.155} C_VEL
LIN {X 0,Y 608.516,Z 562.671,A -85,B 0,C 180,E1 -437.832,E2 -437.832} C_VEL
LIN {X 0,Y 608.499,Z 575.463,A -85,B 0,C 180,E1 -438.676,E2 -438.676} C_VEL
LIN {X 0,Y 608.496,Z 585.925,A -85,B 0,C 180,E1 -439.518,E2 -439.518} C_VEL
LIN {X 0,Y 608.479,Z 596.329,A -85,B 0,C 180,E1 -440.526,E2 -440.526} C_VEL
LIN {X 0,Y 608.464,Z 604.909,A -85,B 0,C 180,E1 -441.531,E2 -441.531} C_VEL
LIN {X 0,Y 608.461,Z 613.11,A -85,B 0,C 180,E1 -442.7,E2 -442.7} C_VEL
LIN {X 0,Y 608.443,Z 619.544,A -85,B 0,C 180,E1 -443.831,E2 -443.831} C_VEL
LIN {X 0,Y 608.438,Z 624.96,A -85,B 0,C 180,E1 -445.03,E2 -445.03} C_VEL
LIN {X 0,Y 608.432,Z 628.439,A -85,B 0,C 180,E1 -446.025,E2 -446.025} C_VEL
LIN {X 0,Y 608.424,Z 631.83,A -85,B 0,C 180,E1 -447.351,E2 -447.351} C_VEL
LIN {X 0,Y 608.442,Z 633.83,A -85,B 0,C 180,E1 -448.676,E2 -448.676} C_VEL
LIN {X 0,Y 608.433,Z 634.5,A -85,B 0,C 180,E1 -449.999,E2 -449.999} C_VEL
LIN {X 0,Y 608.442,Z 633.831,A -85,B 0,C 180,E1 -451.323,E2 -451.323} C_VEL
LIN {X 0,Y 608.424,Z 631.832,A -85,B 0,C 180,E1 -452.648,E2 -452.648} C_VEL
LIN {X 0,Y 608.431,Z 628.443,A -85,B 0,C 180,E1 -453.973,E2 -453.973} C_VEL
LIN {X 0,Y 608.44,Z 623.57,A -85,B 0,C 180,E1 -455.301,E2 -455.301} C_VEL
LIN {X 0,Y 608.445,Z 617.214,A -85,B 0,C 180,E1 -456.603,E2 -456.603} C_VEL
LIN {X 0,Y 608.453,Z 609.802,A -85,B 0,C 180,E1 -457.8,E2 -457.8} C_VEL
LIN {X 0,Y 608.472,Z 600.829,A -85,B 0,C 180,E1 -458.97,E2 -458.97} C_VEL
LIN {X 0,Y 608.472,Z 591.398,A -85,B 0,C 180,E1 -459.976,E2 -459.976} C_VEL
LIN {X 0,Y 608.505,Z 580.051,A -85,B 0,C 180,E1 -460.973,E2 -460.973} C_VEL
LIN {X 0,Y 608.533,Z 568.158,A -85,B 0,C 180,E1 -461.829,E2 -461.829} C_VEL
LIN {X 0,Y 608.531,Z 555.085,A -85,B 0,C 180,E1 -462.59,E2 -462.59} C_VEL
LIN {X 0,Y 608.556,Z 542.188,A -85,B 0,C 180,E1 -463.184,E2 -463.184} C_VEL
LIN {X 0,Y 608.593,Z 528.205,A -85,B 0,C 180,E1 -463.672,E2 -463.672} C_VEL
LIN {X 0,Y 608.62,Z 514.489,A -85,B 0,C 180,E1 -464.012,E2 -464.012} C_VEL
LIN {X 0,Y 608.62,Z 498.221,A -85,B 0,C 180,E1 -464.257,E2 -464.257} C_VEL
LIN {X 0,Y 608.524,Z 371.423,A -85,B 0,C 180,E1 -465.78,E2 -465.78} C_VEL
LIN {X 0,Y 608.563,Z 346.655,A -85,B 0,C 180,E1 -468.741,E2 -468.741} C_VEL
LIN {X 0,Y 608.588,Z 322.456,A -85,B 0,C 180,E1 -471.686,E2 -471.686} C_VEL
LIN {X 0,Y 608.541,Z 303.719,A -85,B 0,C 180,E1 -474.011,E2 -474.011} C_VEL
LIN {X 0,Y 608.461,Z 303.314,A -85,B 0,C 180,E1 -474.071,E2 -474.071} C_VEL
LIN {X 0,Y 608.445,Z 303.319,A -85,B 0,C 180,E1 -476.774,E2 -476.774} C_VEL
LIN {X 0,Y 608.481,Z 303.31,A -85,B 0,C 180,E1 -479.778,E2 -479.778} C_VEL
LIN {X 0,Y 608.448,Z 303.317,A -85,B 0,C 180,E1 -482.52,E2 -482.52} C_VEL
LIN {X 0,Y 608.447,Z 303.317,A -85,B 0,C 180,E1 -485.276,E2 -485.276} C_VEL
LIN {X 0,Y 608.466,Z 303.311,A -85,B 0,C 180,E1 -487.745,E2 -487.745} C_VEL
LIN {X 0,Y 608.447,Z 303.317,A -85,B 0,C 180,E1 -490.328,E2 -490.328} C_VEL
LIN {X 0,Y 608.445,Z 303.32,A -85,B 0,C 180,E1 -492.959,E2 -492.959} C_VEL
LIN {X 0,Y 608.459,Z 303.312,A -85,B 0,C 180,E1 -495.735,E2 -495.735} C_VEL
LIN {X 0,Y 608.463,Z 303.321,A -85,B 0,C 180,E1 -498.656,E2 -498.656} C_VEL
LIN {X 0,Y 608.459,Z 303.312,A -85,B 0,C 180,E1 -501.411,E2 -501.411} C_VEL
LIN {X 0,Y 608.474,Z 303.312,A -85,B 0,C 180,E1 -503.949,E2 -503.949} C_VEL
LIN {X 0,Y 608.469,Z 303.319,A -85,B 0,C 180,E1 -506.329,E2 -506.329} C_VEL
LIN {X 0,Y 608.437,Z 303.319,A -85,B 0,C 180,E1 -508.732,E2 -508.732} C_VEL
LIN {X 0,Y 608.466,Z 303.311,A -85,B 0,C 180,E1 -511.379,E2 -511.379} C_VEL
LIN {X 0,Y 608.474,Z 303.321,A -85,B 0,C 180,E1 -514.276,E2 -514.276} C_VEL
LIN {X 0,Y 608.432,Z 303.316,A -85,B 0,C 180,E1 -516.875,E2 -516.875} C_VEL
LIN {X 0,Y 608.463,Z 303.315,A -85,B 0,C 180,E1 -519.726,E2 -519.726} C_VEL
LIN {X 0,Y 608.431,Z 303.319,A -85,B 0,C 180,E1 -522.523,E2 -522.523} C_VEL
LIN {X 0,Y 608.463,Z 303.312,A -85,B 0,C 180,E1 -525.279,E2 -525.279} C_VEL
LIN {X 0,Y 608.454,Z 303.323,A -85,B 0,C 180,E1 -528,E2 -528} C_VEL
LIN {X 0,Y 608.432,Z 303.316,A -85,B 0,C 180,E1 -530.693,E2 -530.693} C_VEL
LIN {X 0,Y 608.469,Z 303.313,A -85,B 0,C 180,E1 -533.367,E2 -533.367} C_VEL
LIN {X 0,Y 608.435,Z 303.321,A -85,B 0,C 180,E1 -536.026,E2 -536.026} C_VEL
LIN {X 0,Y 608.43,Z 303.321,A -85,B 0,C 180,E1 -538.014,E2 -538.014} C_VEL
LIN {X 0,Y 608.454,Z 303.318,A -85,B 0,C 180,E1 -540,E2 -540} C_VEL
LIN {X 0,Y 608.42,Z 303.316,A -85,B 0,C 180,E1 -542.648,E2 -542.648} C_VEL
LIN {X 0,Y 608.445,Z 303.319,A -85,B 0,C 180,E1 -545.302,E2 -545.302} C_VEL
LIN {X 0,Y 608.415,Z 303.321,A -85,B 0,C 180,E1 -547.968,E2 -547.968} C_VEL
LIN {X 0,Y 608.433,Z 303.32,A -85,B 0,C 180,E1 -549.412,E2 -549.412} C_VEL
LIN {X 0,Y 607.744,Z 303.404,A -85,B 0,C 180,E1 -549.964,E2 -549.964} C_VEL
LIN {X 0,Y 604.891,Z 303.758,A -85,B 0,C 180,E1 -550.861,E2 -550.861} C_VEL
LIN {X 0,Y 602.488,Z 304.064,A -85,B 0,C 180,E1 -551.582,E2 -551.582} C_VEL
LIN {X 0,Y 601.447,Z 304.187,A -85,B 0,C 180,E1 -552.139,E2 -552.139} C_VEL
LIN {X 0,Y 601.357,Z 304.196,A -85,B 0,C 180,E1 -552.327,E2 -552.327} C_VEL
LIN {X 0,Y 601.368,Z 304.198,A -85,B 0,C 180,E1 -554.898,E2 -554.898} C_VEL
LIN {X 0,Y 601.368,Z 304.2,A -85,B 0,C 180,E1 -557.689,E2 -557.689} C_VEL
LIN {X 0,Y 601.373,Z 304.197,A -85,B 0,C 180,E1 -559.81,E2 -559.81} C_VEL
LIN {X 0,Y 601.389,Z 304.194,A -85,B 0,C 180,E1 -562.684,E2 -562.684} C_VEL
LIN {X 0,Y 601.412,Z 304.193,A -85,B 0,C 180,E1 -565.618,E2 -565.618} C_VEL
LIN {X 0,Y 601.356,Z 304.197,A -85,B 0,C 180,E1 -567.87,E2 -567.87} C_VEL
LIN {X 0,Y 601.387,Z 304.193,A -85,B 0,C 180,E1 -570.166,E2 -570.166} C_VEL
LIN {X 0,Y 601.395,Z 304.197,A -85,B 0,C 180,E1 -572.713,E2 -572.713} C_VEL
LIN {X 0,Y 601.384,Z 304.202,A -85,B 0,C 180,E1 -575.112,E2 -575.112} C_VEL
LIN {X 0,Y 601.425,Z 304.191,A -85,B 0,C 180,E1 -577.419,E2 -577.419} C_VEL
LIN {X 0,Y 601.392,Z 304.192,A -85,B 0,C 180,E1 -579.996,E2 -579.996} C_VEL
LIN {X 0,Y 601.401,Z 304.199,A -85,B 0,C 180,E1 -582.671,E2 -582.671} C_VEL
LIN {X 0,Y 601.389,Z 304.193,A -85,B 0,C 180,E1 -585.48,E2 -585.48} C_VEL
LIN {X 0,Y 601.414,Z 304.195,A -85,B 0,C 180,E1 -588.407,E2 -588.407} C_VEL
LIN {X 0,Y 601.43,Z 304.196,A -85,B 0,C 180,E1 -590.876,E2 -590.876} C_VEL
LIN {X 0,Y 601.416,Z 304.235,A -85,B 0,C 180,E1 -591.76,E2 -591.76} C_VEL
LIN {X 0,Y 601.53,Z 317.126,A -85,B 0,C 180,E1 -593.722,E2 -593.722} C_VEL
LIN {X 0,Y 601.476,Z 332.946,A -85,B 0,C 180,E1 -596.095,E2 -596.095} C_VEL
LIN {X 0,Y 601.806,Z 337.335,A -85,B 0,C 180,E1 -596.159,E2 -596.159} C_VEL
LIN {X 0,Y 601.731,Z 469.538,A -85,B 0,C 180,E1 -597.776,E2 -597.776} C_VEL
LIN {X 0,Y 601.684,Z 484,A -85,B 0,C 180,E1 -598.094,E2 -598.094} C_VEL
LIN {X 0,Y 601.65,Z 497.044,A -85,B 0,C 180,E1 -598.509,E2 -598.509} C_VEL
LIN {X 0,Y 601.608,Z 510.303,A -85,B 0,C 180,E1 -599.07,E2 -599.07} C_VEL
LIN {X 0,Y 601.566,Z 523.066,A -85,B 0,C 180,E1 -599.758,E2 -599.758} C_VEL
LIN {X 0,Y 601.506,Z 534.496,A -85,B 0,C 180,E1 -600.516,E2 -600.516} C_VEL
LIN {X 0,Y 601.467,Z 546.286,A -85,B 0,C 180,E1 -601.471,E2 -601.471} C_VEL
LIN {X 0,Y 601.414,Z 555.927,A -85,B 0,C 180,E1 -602.417,E2 -602.417} C_VEL
LIN {X 0,Y 601.419,Z 564.711,A -85,B 0,C 180,E1 -603.451,E2 -603.451} C_VEL
LIN {X 0,Y 601.385,Z 572.543,A -85,B 0,C 180,E1 -604.567,E2 -604.567} C_VEL
LIN {X 0,Y 601.359,Z 579.802,A -85,B 0,C 180,E1 -605.856,E2 -605.856} C_VEL
LIN {X 0,Y 601.352,Z 584.713,A -85,B 0,C 180,E1 -606.952,E2 -606.952} C_VEL
LIN {X 0,Y 601.369,Z 588.492,A -85,B 0,C 180,E1 -608.04,E2 -608.04} C_VEL
LIN {X 0,Y 601.349,Z 592.065,A -85,B 0,C 180,E1 -609.476,E2 -609.476} C_VEL
LIN {X 0,Y 601.312,Z 594.001,A -85,B 0,C 180,E1 -610.898,E2 -610.898} C_VEL
LIN {X 0,Y 601.309,Z 594.445,A -85,B 0,C 180,E1 -612.31,E2 -612.31} C_VEL
LIN {X 0,Y 601.344,Z 593.45,A -85,B 0,C 180,E1 -613.711,E2 -613.711} C_VEL
LIN {X 0,Y 601.315,Z 591.027,A -85,B 0,C 180,E1 -615.101,E2 -615.101} C_VEL
LIN {X 0,Y 601.338,Z 587.123,A -85,B 0,C 180,E1 -616.483,E2 -616.483} C_VEL
LIN {X 0,Y 601.372,Z 583.123,A -85,B 0,C 180,E1 -617.515,E2 -617.515} C_VEL
LIN {X 0,Y 601.364,Z 578.209,A -85,B 0,C 180,E1 -618.541,E2 -618.541} C_VEL
LIN {X 0,Y 601.39,Z 571.141,A -85,B 0,C 180,E1 -619.735,E2 -619.735} C_VEL
LIN {X 0,Y 601.428,Z 562.423,A -85,B 0,C 180,E1 -620.924,E2 -620.924} C_VEL
LIN {X 0,Y 601.452,Z 553.365,A -85,B 0,C 180,E1 -621.94,E2 -621.94} C_VEL
LIN {X 0,Y 601.476,Z 542.458,A -85,B 0,C 180,E1 -622.953,E2 -622.953} C_VEL
LIN {X 0,Y 601.529,Z 530.445,A -85,B 0,C 180,E1 -623.86,E2 -623.86} C_VEL
LIN {X 0,Y 601.567,Z 517.75,A -85,B 0,C 180,E1 -624.638,E2 -624.638} C_VEL
LIN {X 0,Y 601.612,Z 505.814,A -85,B 0,C 180,E1 -625.226,E2 -625.226} C_VEL
LIN {X 0,Y 601.688,Z 492.745,A -85,B 0,C 180,E1 -625.73,E2 -625.73} C_VEL
LIN {X 0,Y 601.7,Z 478.675,A -85,B 0,C 180,E1 -626.129,E2 -626.129} C_VEL
LIN {X 0,Y 601.759,Z 465.008,A -85,B 0,C 180,E1 -626.381,E2 -626.381} C_VEL
LIN {X 0,Y 601.691,Z 334.239,A -85,B 0,C 180,E1 -627.972,E2 -627.972} C_VEL
LIN {X 0,Y 601.497,Z 332.825,A -85,B 0,C 180,E1 -628.013,E2 -628.013} C_VEL
LIN {X 0,Y 601.553,Z 312.912,A -85,B 0,C 180,E1 -631.005,E2 -631.005} C_VEL
LIN {X 0,Y 601.403,Z 304.194,A -85,B 0,C 180,E1 -632.345,E2 -632.345} C_VEL
LIN {X 0,Y 601.402,Z 304.192,A -85,B 0,C 180,E1 -634.693,E2 -634.693} C_VEL
LIN {X 0,Y 601.447,Z 304.196,A -85,B 0,C 180,E1 -637.386,E2 -637.386} C_VEL
LIN {X 0,Y 601.384,Z 304.194,A -85,B 0,C 180,E1 -640.096,E2 -640.096} C_VEL
LIN {X 0,Y 601.391,Z 304.192,A -85,B 0,C 180,E1 -642.144,E2 -642.144} C_VEL
LIN {X 0,Y 601.397,Z 304.196,A -85,B 0,C 180,E1 -644.898,E2 -644.898} C_VEL
LIN {X 0,Y 601.376,Z 304.197,A -85,B 0,C 180,E1 -647.689,E2 -647.689} C_VEL
LIN {X 0,Y 601.381,Z 304.195,A -85,B 0,C 180,E1 -649.811,E2 -649.811} C_VEL
LIN {X 0,Y 601.401,Z 304.193,A -85,B 0,C 180,E1 -652.603,E2 -652.603} C_VEL
LIN {X 0,Y 601.385,Z 304.2,A -85,B 0,C 180,E1 -654.88,E2 -654.88} C_VEL
LIN {X 0,Y 601.393,Z 304.197,A -85,B 0,C 180,E1 -657.359,E2 -657.359} C_VEL
LIN {X 0,Y 601.37,Z 304.199,A -85,B 0,C 180,E1 -659.396,E2 -659.396} C_VEL
LIN {X 0,Y 601.376,Z 304.194,A -85,B 0,C 180,E1 -661.729,E2 -661.729} C_VEL
LIN {X 0,Y 601.379,Z 304.194,A -85,B 0,C 180,E1 -664.122,E2 -664.122} C_VEL
LIN {X 0,Y 601.383,Z 304.198,A -85,B 0,C 180,E1 -666.585,E2 -666.585} C_VEL
LIN {X 0,Y 601.381,Z 304.194,A -85,B 0,C 180,E1 -669.529,E2 -669.529} C_VEL
LIN {X 0,Y 601.368,Z 304.195,A -85,B 0,C 180,E1 -671.77,E2 -671.77} C_VEL
LIN {X 0,Y 601.366,Z 304.202,A -85,B 0,C 180,E1 -674.53,E2 -674.53} C_VEL
LIN {X 0,Y 601.405,Z 304.196,A -85,B 0,C 180,E1 -676.43,E2 -676.43} C_VEL
LIN {X 0,Y 601.381,Z 304.194,A -85,B 0,C 180,E1 -679.431,E2 -679.431} C_VEL
LIN {X 0,Y 601.343,Z 304.198,A -85,B 0,C 180,E1 -681.727,E2 -681.727} C_VEL
LIN {X 0,Y 601.358,Z 304.201,A -85,B 0,C 180,E1 -684.244,E2 -684.244} C_VEL
LIN {X 0,Y 601.407,Z 304.198,A -85,B 0,C 180,E1 -686.686,E2 -686.686} C_VEL
LIN {X 0,Y 601.387,Z 304.195,A -85,B 0,C 180,E1 -689.057,E2 -689.057} C_VEL
LIN {X 0,Y 601.385,Z 304.193,A -85,B 0,C 180,E1 -691.371,E2 -691.371} C_VEL
LIN {X 0,Y 601.397,Z 304.197,A -85,B 0,C 180,E1 -694.136,E2 -694.136} C_VEL
LIN {X 0,Y 601.378,Z 304.201,A -85,B 0,C 180,E1 -696.588,E2 -696.588} C_VEL
LIN {X 0,Y 601.394,Z 304.192,A -85,B 0,C 180,E1 -699.477,E2 -699.477} C_VEL
LIN {X 0,Y 601.368,Z 304.196,A -85,B 0,C 180,E1 -701.607,E2 -701.607} C_VEL
LIN {X 0,Y 601.401,Z 304.199,A -85,B 0,C 180,E1 -704.409,E2 -704.409} C_VEL
LIN {X 0,Y 601.371,Z 304.194,A -85,B 0,C 180,E1 -707.171,E2 -707.171} C_VEL
LIN {X 0,Y 601.427,Z 304.194,A -85,B 0,C 180,E1 -709.905,E2 -709.905} C_VEL
LIN {X 0,Y 601.406,Z 304.193,A -85,B 0,C 180,E1 -712.615,E2 -712.615} C_VEL
LIN {X 0,Y 601.391,Z 304.193,A -85,B 0,C 180,E1 -715.308,E2 -715.308} C_VEL
LIN {X 0,Y 601.434,Z 304.197,A -85,B 0,C 180,E1 -717.991,E2 -717.991} C_VEL
LIN {X 0,Y 601.445,Z 304.186,A -85,B 0,C 180,E1 -720.67,E2 -720.67} C_VEL
LIN {X 0,Y 601.378,Z 304.196,A -85,B 0,C 180,E1 -723.35,E2 -723.35} C_VEL
LIN {X 0,Y 601.421,Z 304.196,A -85,B 0,C 180,E1 -726.037,E2 -726.037} C_VEL
LIN {X 0,Y 601.408,Z 304.19,A -85,B 0,C 180,E1 -728.738,E2 -728.738} C_VEL
LIN {X 0,Y 601.421,Z 304.189,A -85,B 0,C 180,E1 -731.009,E2 -731.009} C_VEL
LIN {X 0,Y 601.425,Z 304.193,A -85,B 0,C 180,E1 -734.092,E2 -734.092} C_VEL
LIN {X 0,Y 601.411,Z 304.19,A -85,B 0,C 180,E1 -736.987,E2 -736.987} C_VEL
LIN {X 0,Y 601.402,Z 304.199,A -85,B 0,C 180,E1 -739.81,E2 -739.81} C_VEL
LIN {X 0,Y 601.414,Z 304.189,A -85,B 0,C 180,E1 -742.683,E2 -742.683} C_VEL
LIN {X 0,Y 601.4,Z 304.192,A -85,B 0,C 180,E1 -744.879,E2 -744.879} C_VEL
LIN {X 0,Y 601.41,Z 304.197,A -85,B 0,C 180,E1 -747.361,E2 -747.361} C_VEL
LIN {X 0,Y 601.431,Z 304.188,A -85,B 0,C 180,E1 -750.164,E2 -750.164} C_VEL
LIN {X 0,Y 601.424,Z 304.189,A -85,B 0,C 180,E1 -752.715,E2 -752.715} C_VEL
LIN {X 0,Y 601.391,Z 304.197,A -85,B 0,C 180,E1 -755.111,E2 -755.111} C_VEL
LIN {X 0,Y 601.437,Z 304.196,A -85,B 0,C 180,E1 -757.419,E2 -757.419} C_VEL
LIN {X 0,Y 601.404,Z 304.192,A -85,B 0,C 180,E1 -759.996,E2 -759.996} C_VEL
LIN {X 0,Y 601.415,Z 304.191,A -85,B 0,C 180,E1 -762.67,E2 -762.67} C_VEL
LIN {X 0,Y 601.402,Z 304.197,A -85,B 0,C 180,E1 -765.479,E2 -765.479} C_VEL
LIN {X 0,Y 601.423,Z 304.189,A -85,B 0,C 180,E1 -768.407,E2 -768.407} C_VEL
LIN {X 0,Y 601.438,Z 304.192,A -85,B 0,C 180,E1 -770.875,E2 -770.875} C_VEL
LIN {X 0,Y 601.404,Z 304.196,A -85,B 0,C 180,E1 -773.417,E2 -773.417} C_VEL
LIN {X 0,Y 601.435,Z 304.187,A -85,B 0,C 180,E1 -776.064,E2 -776.064} C_VEL
LIN {X 0,Y 601.422,Z 304.192,A -85,B 0,C 180,E1 -778.545,E2 -778.545} C_VEL
LIN {X 0,Y 601.421,Z 304.193,A -85,B 0,C 180,E1 -781.372,E2 -781.372} C_VEL
LIN {X 0,Y 601.4,Z 304.193,A -85,B 0,C 180,E1 -783.636,E2 -783.636} C_VEL
LIN {X 0,Y 601.457,Z 304.328,A -85,B 0,C 180,E1 -785.766,E2 -785.766} C_VEL
LIN {X 0,Y 601.775,Z 307.963,A -85,B 0,C 180,E1 -786.239,E2 -786.239} C_VEL
LIN {X 0,Y 601.692,Z 330.416,A -85,B 0,C 180,E1 -789.041,E2 -789.041} C_VEL
LIN {X 0,Y 601.617,Z 352.857,A -85,B 0,C 180,E1 -791.79,E2 -791.79} C_VEL
LIN {X 0,Y 601.543,Z 371.412,A -85,B 0,C 180,E1 -794.031,E2 -794.031} C_VEL
LIN {X 0,Y 601.831,Z 377.363,A -85,B 0,C 180,E1 -794.115,E2 -794.115} C_VEL
LIN {X 0,Y 601.734,Z 509.954,A -85,B 0,C 180,E1 -795.739,E2 -795.739} C_VEL
LIN {X 0,Y 601.698,Z 523.896,A -85,B 0,C 180,E1 -796.046,E2 -796.046} C_VEL
LIN {X 0,Y 601.651,Z 537.699,A -85,B 0,C 180,E1 -796.489,E2 -796.489} C_VEL
LIN {X 0,Y 601.609,Z 551.623,A -85,B 0,C 180,E1 -797.09,E2 -797.09} C_VEL
LIN {X 0,Y 601.547,Z 564.085,A -85,B 0,C 180,E1 -797.774,E2 -797.774} C_VEL
LIN {X 0,Y 601.505,Z 575.465,A -85,B 0,C 180,E1 -798.543,E2 -798.543} C_VEL
LIN {X 0,Y 601.482,Z 585.926,A -85,B 0,C 180,E1 -799.395,E2 -799.395} C_VEL
LIN {X 0,Y 601.43,Z 596.329,A -85,B 0,C 180,E1 -800.414,E2 -800.414} C_VEL
LIN {X 0,Y 601.407,Z 604.909,A -85,B 0,C 180,E1 -801.431,E2 -801.431} C_VEL
LIN {X 0,Y 601.392,Z 613.111,A -85,B 0,C 180,E1 -802.614,E2 -802.614} C_VEL
LIN {X 0,Y 601.361,Z 618.751,A -85,B 0,C 180,E1 -803.604,E2 -803.604} C_VEL
LIN {X 0,Y 601.355,Z 623.565,A -85,B 0,C 180,E1 -804.635,E2 -804.635} C_VEL
LIN {X 0,Y 601.343,Z 628.44,A -85,B 0,C 180,E1 -805.978,E2 -805.978} C_VEL
LIN {X 0,Y 601.324,Z 631.83,A -85,B 0,C 180,E1 -807.32,E2 -807.32} C_VEL
LIN {X 0,Y 601.342,Z 633.83,A -85,B 0,C 180,E1 -808.66,E2 -808.66} C_VEL
LIN {X 0,Y 601.333,Z 634.5,A -85,B 0,C 180,E1 -809.999,E2 -809.999} C_VEL
LIN {X 0,Y 601.342,Z 633.832,A -85,B 0,C 180,E1 -811.339,E2 -811.339} C_VEL
LIN {X 0,Y 601.324,Z 631.833,A -85,B 0,C 180,E1 -812.679,E2 -812.679} C_VEL
LIN {X 0,Y 601.343,Z 628.444,A -85,B 0,C 180,E1 -814.02,E2 -814.02} C_VEL
LIN {X 0,Y 601.355,Z 623.57,A -85,B 0,C 180,E1 -815.364,E2 -815.364} C_VEL
LIN {X 0,Y 601.354,Z 617.055,A -85,B 0,C 180,E1 -816.711,E2 -816.711} C_VEL
LIN {X 0,Y 601.398,Z 609.803,A -85,B 0,C 180,E1 -817.892,E2 -817.892} C_VEL
LIN {X 0,Y 601.43,Z 600.829,A -85,B 0,C 180,E1 -819.076,E2 -819.076} C_VEL
LIN {X 0,Y 601.44,Z 591.398,A -85,B 0,C 180,E1 -820.094,E2 -820.094} C_VEL
LIN {X 0,Y 601.504,Z 580.698,A -85,B 0,C 180,E1 -821.05,E2 -821.05} C_VEL
LIN {X 0,Y 601.544,Z 569.437,A -85,B 0,C 180,E1 -821.883,E2 -821.883} C_VEL
LIN {X 0,Y 601.565,Z 556.657,A -85,B 0,C 180,E1 -822.653,E2 -822.653} C_VEL
LIN {X 0,Y 601.626,Z 544.175,A -85,B 0,C 180,E1 -823.252,E2 -823.252} C_VEL
LIN {X 0,Y 601.69,Z 530.845,A -85,B 0,C 180,E1 -823.748,E2 -823.748} C_VEL
LIN {X 0,Y 601.733,Z 516.541,A -85,B 0,C 180,E1 -824.133,E2 -824.133} C_VEL
LIN {X 0,Y 601.743,Z 502.152,A -85,B 0,C 180,E1 -824.376,E2 -824.376} C_VEL
LIN {X 0,Y 601.736,Z 372.771,A -85,B 0,C 180,E1 -825.943,E2 -825.943} C_VEL
LIN {X 0,Y 601.549,Z 371.332,A -85,B 0,C 180,E1 -825.978,E2 -825.978} C_VEL
LIN {X 0,Y 601.628,Z 347.379,A -85,B 0,C 180,E1 -828.877,E2 -828.877} C_VEL
LIN {X 0,Y 601.689,Z 323.904,A -85,B 0,C 180,E1 -831.767,E2 -831.767} C_VEL
LIN {X 0,Y 601.795,Z 306.525,A -85,B 0,C 180,E1 -833.942,E2 -833.942} C_VEL
LIN {X 0,Y 601.419,Z 304.194,A -85,B 0,C 180,E1 -834.255,E2 -834.255} C_VEL
LIN {X 0,Y 601.455,Z 304.194,A -85,B 0,C 180,E1 -837.11,E2 -837.11} C_VEL
LIN {X 0,Y 601.427,Z 304.188,A -85,B 0,C 180,E1 -840.148,E2 -840.148} C_VEL
LIN {X 0,Y 601.412,Z 304.196,A -85,B 0,C 180,E1 -842.714,E2 -842.714} C_VEL
LIN {X 0,Y 601.414,Z 304.196,A -85,B 0,C 180,E1 -845.114,E2 -845.114} C_VEL
LIN {X 0,Y 601.432,Z 304.189,A -85,B 0,C 180,E1 -847.418,E2 -847.418} C_VEL
LIN {X 0,Y 601.408,Z 304.191,A -85,B 0,C 180,E1 -849.994,E2 -849.994} C_VEL
LIN {X 0,Y 601.406,Z 304.2,A -85,B 0,C 180,E1 -852.67,E2 -852.67} C_VEL
LIN {X 0,Y 601.421,Z 304.188,A -85,B 0,C 180,E1 -855.481,E2 -855.481} C_VEL
LIN {X 0,Y 601.424,Z 304.195,A -85,B 0,C 180,E1 -858.405,E2 -858.405} C_VEL
LIN {X 0,Y 601.426,Z 304.192,A -85,B 0,C 180,E1 -860.874,E2 -860.874} C_VEL
LIN {X 0,Y 601.437,Z 304.187,A -85,B 0,C 180,E1 -863.733,E2 -863.733} C_VEL
LIN {X 0,Y 601.426,Z 304.194,A -85,B 0,C 180,E1 -866.686,E2 -866.686} C_VEL
LIN {X 0,Y 601.443,Z 304.188,A -85,B 0,C 180,E1 -869.847,E2 -869.847} C_VEL
LIN {X 0,Y 601.401,Z 304.195,A -85,B 0,C 180,E1 -872.638,E2 -872.638} C_VEL
LIN {X 0,Y 601.391,Z 304.192,A -85,B 0,C 180,E1 -875.121,E2 -875.121} C_VEL
LIN {X 0,Y 601.407,Z 304.19,A -85,B 0,C 180,E1 -877.394,E2 -877.394} C_VEL
LIN {X 0,Y 601.396,Z 304.201,A -85,B 0,C 180,E1 -880.19,E2 -880.19} C_VEL
LIN {X 0,Y 601.384,Z 304.2,A -85,B 0,C 180,E1 -882.311,E2 -882.311} C_VEL
LIN {X 0,Y 601.395,Z 304.196,A -85,B 0,C 180,E1 -884.408,E2 -884.408} C_VEL
LIN {X 0,Y 601.403,Z 304.191,A -85,B 0,C 180,E1 -887.171,E2 -887.171} C_VEL
LIN {X 0,Y 601.423,Z 304.198,A -85,B 0,C 180,E1 -889.905,E2 -889.905} C_VEL
LIN {X 0,Y 601.385,Z 304.193,A -85,B 0,C 180,E1 -892.614,E2 -892.614} C_VEL
LIN {X 0,Y 601.414,Z 304.192,A -85,B 0,C 180,E1 -895.308,E2 -895.308} C_VEL
LIN {X 0,Y 601.402,Z 304.197,A -85,B 0,C 180,E1 -897.991,E2 -897.991} C_VEL
LIN {X 0,Y 601.424,Z 304.194,A -85,B 0,C 180,E1 -900,E2 -900} C_VEL
LIN {X 0,Y 601.391,Z 304.192,A -85,B 0,C 180,E1 -902.679,E2 -902.679} C_VEL
LIN {X 0,Y 601.408,Z 304.196,A -85,B 0,C 180,E1 -905.364,E2 -905.364} C_VEL
LIN {X 0,Y 601.386,Z 304.195,A -85,B 0,C 180,E1 -908.061,E2 -908.061} C_VEL
LIN {X 0,Y 601.386,Z 304.196,A -85,B 0,C 180,E1 -910.998,E2 -910.998} C_VEL
LIN {X 0,Y 601.357,Z 304.196,A -85,B 0,C 180,E1 -912.327,E2 -912.327} C_VEL
LIN {X 0,Y 600.677,Z 304.284,A -85,B 0,C 180,E1 -912.886,E2 -912.886} C_VEL
LIN {X 0,Y 597.83,Z 304.64,A -85,B 0,C 180,E1 -913.794,E2 -913.794} C_VEL
LIN {X 0,Y 595.432,Z 304.94,A -85,B 0,C 180,E1 -914.524,E2 -914.524} C_VEL
LIN {X 0,Y 594.401,Z 305.068,A -85,B 0,C 180,E1 -915.088,E2 -915.088} C_VEL
LIN {X 0,Y 594.315,Z 305.077,A -85,B 0,C 180,E1 -915.279,E2 -915.279} C_VEL
LIN {X 0,Y 594.313,Z 305.076,A -85,B 0,C 180,E1 -917.906,E2 -917.906} C_VEL
LIN {X 0,Y 594.365,Z 305.07,A -85,B 0,C 180,E1 -920.777,E2 -920.777} C_VEL
LIN {X 0,Y 594.334,Z 305.074,A -85,B 0,C 180,E1 -923.706,E2 -923.706} C_VEL
LIN {X 0,Y 594.355,Z 305.069,A -85,B 0,C 180,E1 -926.019,E2 -926.019} C_VEL
LIN {X 0,Y 594.315,Z 305.073,A -85,B 0,C 180,E1 -928.23,E2 -928.23} C_VEL
LIN {X 0,Y 594.357,Z 305.071,A -85,B 0,C 180,E1 -930.561,E2 -930.561} C_VEL
LIN {X 0,Y 594.363,Z 305.077,A -85,B 0,C 180,E1 -932.951,E2 -932.951} C_VEL
LIN {X 0,Y 594.338,Z 305.075,A -85,B 0,C 180,E1 -935.409,E2 -935.409} C_VEL
LIN {X 0,Y 594.364,Z 305.068,A -85,B 0,C 180,E1 -937.942,E2 -937.942} C_VEL
LIN {X 0,Y 594.368,Z 305.077,A -85,B 0,C 180,E1 -940.822,E2 -940.822} C_VEL
LIN {X 0,Y 594.351,Z 305.069,A -85,B 0,C 180,E1 -943.839,E2 -943.839} C_VEL
LIN {X 0,Y 594.358,Z 305.078,A -85,B 0,C 180,E1 -946.701,E2 -946.701} C_VEL
LIN {X 0,Y 594.356,Z 305.07,A -85,B 0,C 180,E1 -949.433,E2 -949.433} C_VEL
LIN {X 0,Y 594.388,Z 305.19,A -85,B 0,C 180,E1 -951.657,E2 -951.657} C_VEL
LIN {X 0,Y 594.551,Z 315.476,A -85,B 0,C 180,E1 -953.247,E2 -953.247} C_VEL
LIN {X 0,Y 594.478,Z 332.874,A -85,B 0,C 180,E1 -955.891,E2 -955.891} C_VEL
LIN {X 0,Y 594.979,Z 337.294,A -85,B 0,C 180,E1 -955.971,E2 -955.971} C_VEL
LIN {X 0,Y 594.858,Z 469.593,A -85,B 0,C 180,E1 -957.608,E2 -957.608} C_VEL
LIN {X 0,Y 594.814,Z 483.985,A -85,B 0,C 180,E1 -957.929,E2 -957.929} C_VEL
LIN {X 0,Y 594.746,Z 498.051,A -85,B 0,C 180,E1 -958.388,E2 -958.388} C_VEL
LIN {X 0,Y 594.674,Z 511.305,A -85,B 0,C 180,E1 -958.965,E2 -958.965} C_VEL
LIN {X 0,Y 594.601,Z 523.466,A -85,B 0,C 180,E1 -959.636,E2 -959.636} C_VEL
LIN {X 0,Y 594.515,Z 535.146,A -85,B 0,C 180,E1 -960.427,E2 -960.427} C_VEL
LIN {X 0,Y 594.459,Z 546.827,A -85,B 0,C 180,E1 -961.393,E2 -961.393} C_VEL
LIN {X 0,Y 594.38,Z 557.48,A -85,B 0,C 180,E1 -962.474,E2 -962.474} C_VEL
LIN {X 0,Y 594.341,Z 565.761,A -85,B 0,C 180,E1 -963.488,E2 -963.488} C_VEL
LIN {X 0,Y 594.31,Z 573.391,A -85,B 0,C 180,E1 -964.618,E2 -964.618} C_VEL
LIN {X 0,Y 594.279,Z 578.836,A -85,B 0,C 180,E1 -965.589,E2 -965.589} C_VEL
LIN {X 0,Y 594.271,Z 583.756,A -85,B 0,C 180,E1 -966.661,E2 -966.661} C_VEL
LIN {X 0,Y 594.262,Z 588.919,A -85,B 0,C 180,E1 -968.129,E2 -968.129} C_VEL
LIN {X 0,Y 594.25,Z 591.592,A -85,B 0,C 180,E1 -969.22,E2 -969.22} C_VEL
LIN {X 0,Y 594.21,Z 593.799,A -85,B 0,C 180,E1 -970.661,E2 -970.661} C_VEL
LIN {X 0,Y 594.25,Z 594.339,A -85,B 0,C 180,E1 -971.379,E2 -971.379} C_VEL
LIN {X 0,Y 594.235,Z 594.277,A -85,B 0,C 180,E1 -972.803,E2 -972.803} C_VEL
LIN {X 0,Y 594.25,Z 592.775,A -85,B 0,C 180,E1 -974.217,E2 -974.217} C_VEL
LIN {X 0,Y 594.236,Z 589.833,A -85,B 0,C 180,E1 -975.62,E2 -975.62} C_VEL
LIN {X 0,Y 594.258,Z 585.393,A -85,B 0,C 180,E1 -977.015,E2 -977.015} C_VEL
LIN {X 0,Y 594.266,Z 580.994,A -85,B 0,C 180,E1 -978.056,E2 -978.056} C_VEL
LIN {X 0,Y 594.286,Z 574.614,A -85,B 0,C 180,E1 -979.266,E2 -979.266} C_VEL
LIN {X 0,Y 594.321,Z 566.705,A -85,B 0,C 180,E1 -980.471,E2 -980.471} C_VEL
LIN {X 0,Y 594.358,Z 558.482,A -85,B 0,C 180,E1 -981.501,E2 -981.501} C_VEL
LIN {X 0,Y 594.455,Z 548.62,A -85,B 0,C 180,E1 -982.528,E2 -982.528} C_VEL
LIN {X 0,Y 594.534,Z 537.56,A -85,B 0,C 180,E1 -983.481,E2 -983.481} C_VEL
LIN {X 0,Y 594.553,Z 525.68,A -85,B 0,C 180,E1 -984.319,E2 -984.319} C_VEL
LIN {X 0,Y 594.646,Z 513.82,A -85,B 0,C 180,E1 -985,E2 -985} C_VEL
LIN {X 0,Y 594.723,Z 500.822,A -85,B 0,C 180,E1 -985.595,E2 -985.595} C_VEL
LIN {X 0,Y 594.786,Z 486.707,A -85,B 0,C 180,E1 -986.084,E2 -986.084} C_VEL
LIN {X 0,Y 594.862,Z 472.63,A -85,B 0,C 180,E1 -986.423,E2 -986.423} C_VEL
LIN {X 0,Y 594.874,Z 453.279,A -85,B 0,C 180,E1 -986.699,E2 -986.699} C_VEL
LIN {X 0,Y 594.862,Z 335.053,A -85,B 0,C 180,E1 -988.149,E2 -988.149} C_VEL
LIN {X 0,Y 594.478,Z 332.86,A -85,B 0,C 180,E1 -988.201,E2 -988.201} C_VEL
LIN {X 0,Y 594.585,Z 314.34,A -85,B 0,C 180,E1 -991.017,E2 -991.017} C_VEL
LIN {X 0,Y 594.394,Z 305.308,A -85,B 0,C 180,E1 -992.415,E2 -992.415} C_VEL
LIN {X 0,Y 594.383,Z 305.07,A -85,B 0,C 180,E1 -992.542,E2 -992.542} C_VEL
LIN {X 0,Y 594.39,Z 305.075,A -85,B 0,C 180,E1 -995.428,E2 -995.428} C_VEL
LIN {X 0,Y 594.348,Z 305.071,A -85,B 0,C 180,E1 -998.158,E2 -998.158} C_VEL
LIN {X 0,Y 594.382,Z 305.072,A -85,B 0,C 180,E1 -1001.071,E2 -1001.071} C_VEL
LIN {X 0,Y 594.36,Z 305.072,A -85,B 0,C 180,E1 -1003.68,E2 -1003.68} C_VEL
LIN {X 0,Y 594.358,Z 305.071,A -85,B 0,C 180,E1 -1006.708,E2 -1006.708} C_VEL
LIN {X 0,Y 594.355,Z 305.076,A -85,B 0,C 180,E1 -1009.335,E2 -1009.335} C_VEL
LIN {X 0,Y 594.345,Z 305.074,A -85,B 0,C 180,E1 -1011.505,E2 -1011.505} C_VEL
LIN {X 0,Y 594.339,Z 305.072,A -85,B 0,C 180,E1 -1014.449,E2 -1014.449} C_VEL
LIN {X 0,Y 594.366,Z 305.072,A -85,B 0,C 180,E1 -1016.701,E2 -1016.701} C_VEL
LIN {X 0,Y 594.367,Z 305.078,A -85,B 0,C 180,E1 -1019,E2 -1019} C_VEL
LIN {X 0,Y 594.352,Z 305.07,A -85,B 0,C 180,E1 -1021.639,E2 -1021.639} C_VEL
LIN {X 0,Y 594.364,Z 305.072,A -85,B 0,C 180,E1 -1024.581,E2 -1024.581} C_VEL
LIN {X 0,Y 594.343,Z 305.071,A -85,B 0,C 180,E1 -1027.603,E2 -1027.603} C_VEL
LIN {X 0,Y 594.351,Z 305.075,A -85,B 0,C 180,E1 -1030.569,E2 -1030.569} C_VEL
LIN {X 0,Y 594.319,Z 305.075,A -85,B 0,C 180,E1 -1033.304,E2 -1033.304} C_VEL
LIN {X 0,Y 594.332,Z 305.074,A -85,B 0,C 180,E1 -1036.165,E2 -1036.165} C_VEL
LIN {X 0,Y 594.354,Z 305.071,A -85,B 0,C 180,E1 -1039.181,E2 -1039.181} C_VEL
LIN {X 0,Y 594.303,Z 305.077,A -85,B 0,C 180,E1 -1042.053,E2 -1042.053} C_VEL
LIN {X 0,Y 594.31,Z 305.083,A -85,B 0,C 180,E1 -1044.683,E2 -1044.683} C_VEL
LIN {X 0,Y 594.367,Z 305.069,A -85,B 0,C 180,E1 -1047.091,E2 -1047.091} C_VEL
LIN {X 0,Y 594.346,Z 305.07,A -85,B 0,C 180,E1 -1049.679,E2 -1049.679} C_VEL
LIN {X 0,Y 594.358,Z 305.077,A -85,B 0,C 180,E1 -1052.539,E2 -1052.539} C_VEL
LIN {X 0,Y 594.362,Z 305.072,A -85,B 0,C 180,E1 -1054.807,E2 -1054.807} C_VEL
LIN {X 0,Y 594.308,Z 305.074,A -85,B 0,C 180,E1 -1057.278,E2 -1057.278} C_VEL
LIN {X 0,Y 594.352,Z 305.073,A -85,B 0,C 180,E1 -1059.946,E2 -1059.946} C_VEL
LIN {X 0,Y 594.33,Z 305.074,A -85,B 0,C 180,E1 -1062.805,E2 -1062.805} C_VEL
LIN {X 0,Y 594.354,Z 305.07,A -85,B 0,C 180,E1 -1065.622,E2 -1065.622} C_VEL
LIN {X 0,Y 594.377,Z 305.072,A -85,B 0,C 180,E1 -1068.404,E2 -1068.404} C_VEL
LIN {X 0,Y 594.361,Z 305.068,A -85,B 0,C 180,E1 -1071.158,E2 -1071.158} C_VEL
LIN {X 0,Y 594.363,Z 305.074,A -85,B 0,C 180,E1 -1073.891,E2 -1073.891} C_VEL
LIN {X 0,Y 594.373,Z 305.068,A -85,B 0,C 180,E1 -1076.611,E2 -1076.611} C_VEL
LIN {X 0,Y 594.397,Z 305.064,A -85,B 0,C 180,E1 -1079.323,E2 -1079.323} C_VEL
LIN {X 0,Y 594.406,Z 305.071,A -85,B 0,C 180,E1 -1082.033,E2 -1082.033} C_VEL
LIN {X 0,Y 594.388,Z 305.065,A -85,B 0,C 180,E1 -1084.748,E2 -1084.748} C_VEL
LIN {X 0,Y 594.368,Z 305.071,A -85,B 0,C 180,E1 -1087.474,E2 -1087.474} C_VEL
LIN {X 0,Y 594.398,Z 305.067,A -85,B 0,C 180,E1 -1090.216,E2 -1090.216} C_VEL
LIN {X 0,Y 594.358,Z 305.069,A -85,B 0,C 180,E1 -1092.983,E2 -1092.983} C_VEL
LIN {X 0,Y 594.368,Z 305.068,A -85,B 0,C 180,E1 -1095.078,E2 -1095.078} C_VEL
LIN {X 0,Y 594.377,Z 305.068,A -85,B 0,C 180,E1 -1097.194,E2 -1097.194} C_VEL
LIN {X 0,Y 594.373,Z 305.07,A -85,B 0,C 180,E1 -1100.054,E2 -1100.054} C_VEL
LIN {X 0,Y 594.358,Z 305.07,A -85,B 0,C 180,E1 -1102.968,E2 -1102.968} C_VEL
LIN {X 0,Y 594.377,Z 305.07,A -85,B 0,C 180,E1 -1105.193,E2 -1105.193} C_VEL
LIN {X 0,Y 594.371,Z 305.077,A -85,B 0,C 180,E1 -1107.523,E2 -1107.523} C_VEL
LIN {X 0,Y 594.388,Z 305.065,A -85,B 0,C 180,E1 -1110.328,E2 -1110.328} C_VEL
LIN {X 0,Y 594.382,Z 305.068,A -85,B 0,C 180,E1 -1112.95,E2 -1112.95} C_VEL
LIN {X 0,Y 594.351,Z 305.08,A -85,B 0,C 180,E1 -1115.409,E2 -1115.409} C_VEL
LIN {X 0,Y 594.386,Z 305.067,A -85,B 0,C 180,E1 -1117.941,E2 -1117.941} C_VEL
LIN {X 0,Y 594.378,Z 305.069,A -85,B 0,C 180,E1 -1120.822,E2 -1120.822} C_VEL
LIN {X 0,Y 594.371,Z 305.077,A -85,B 0,C 180,E1 -1123.299,E2 -1123.299} C_VEL
LIN {X 0,Y 594.363,Z 305.068,A -85,B 0,C 180,E1 -1126.161,E2 -1126.161} C_VEL
LIN {X 0,Y 594.381,Z 305.067,A -85,B 0,C 180,E1 -1128.536,E2 -1128.536} C_VEL
LIN {X 0,Y 594.39,Z 305.072,A -85,B 0,C 180,E1 -1131.295,E2 -1131.295} C_VEL
LIN {X 0,Y 594.354,Z 305.07,A -85,B 0,C 180,E1 -1133.755,E2 -1133.755} C_VEL
LIN {X 0,Y 594.378,Z 305.066,A -85,B 0,C 180,E1 -1136.238,E2 -1136.238} C_VEL
LIN {X 0,Y 594.371,Z 305.072,A -85,B 0,C 180,E1 -1138.649,E2 -1138.649} C_VEL
LIN {X 0,Y 594.384,Z 305.076,A -85,B 0,C 180,E1 -1141.042,E2 -1141.042} C_VEL
LIN {X 0,Y 594.386,Z 305.066,A -85,B 0,C 180,E1 -1143.978,E2 -1143.978} C_VEL
LIN {X 0,Y 594.398,Z 305.151,A -85,B 0,C 180,E1 -1145.565,E2 -1145.565} C_VEL
LIN {X 0,Y 594.929,Z 309.411,A -85,B 0,C 180,E1 -1146.133,E2 -1146.133} C_VEL
LIN {X 0,Y 594.794,Z 331.965,A -85,B 0,C 180,E1 -1148.98,E2 -1148.98} C_VEL
LIN {X 0,Y 594.653,Z 355.754,A -85,B 0,C 180,E1 -1151.926,E2 -1151.926} C_VEL
LIN {X 0,Y 594.549,Z 371.412,A -85,B 0,C 180,E1 -1153.838,E2 -1153.838} C_VEL
LIN {X 0,Y 595.023,Z 375.574,A -85,B 0,C 180,E1 -1153.907,E2 -1153.907} C_VEL
LIN {X 0,Y 594.859,Z 509.858,A -85,B 0,C 180,E1 -1155.569,E2 -1155.569} C_VEL
LIN {X 0,Y 594.816,Z 524.118,A -85,B 0,C 180,E1 -1155.888,E2 -1155.888} C_VEL
LIN {X 0,Y 594.74,Z 537.701,A -85,B 0,C 180,E1 -1156.329,E2 -1156.329} C_VEL
LIN {X 0,Y 594.663,Z 551.625,A -85,B 0,C 180,E1 -1156.936,E2 -1156.936} C_VEL
LIN {X 0,Y 594.582,Z 564.087,A -85,B 0,C 180,E1 -1157.629,E2 -1157.629} C_VEL
LIN {X 0,Y 594.525,Z 576.548,A -85,B 0,C 180,E1 -1158.487,E2 -1158.487} C_VEL
LIN {X 0,Y 594.449,Z 587.831,A -85,B 0,C 180,E1 -1159.44,E2 -1159.44} C_VEL
LIN {X 0,Y 594.368,Z 597.845,A -85,B 0,C 180,E1 -1160.471,E2 -1160.471} C_VEL
LIN {X 0,Y 594.324,Z 606.166,A -85,B 0,C 180,E1 -1161.499,E2 -1161.499} C_VEL
LIN {X 0,Y 594.303,Z 614.122,A -85,B 0,C 180,E1 -1162.696,E2 -1162.696} C_VEL
LIN {X 0,Y 594.279,Z 620.524,A -85,B 0,C 180,E1 -1163.89,E2 -1163.89} C_VEL
LIN {X 0,Y 594.237,Z 626.197,A -85,B 0,C 180,E1 -1165.251,E2 -1165.251} C_VEL
LIN {X 0,Y 594.259,Z 630.314,A -85,B 0,C 180,E1 -1166.609,E2 -1166.609} C_VEL
LIN {X 0,Y 594.24,Z 632.999,A -85,B 0,C 180,E1 -1167.966,E2 -1167.966} C_VEL
LIN {X 0,Y 594.237,Z 634.332,A -85,B 0,C 180,E1 -1169.322,E2 -1169.322} C_VEL
LIN {X 0,Y 594.237,Z 634.333,A -85,B 0,C 180,E1 -1170.677,E2 -1170.677} C_VEL
LIN {X 0,Y 594.24,Z 633.001,A -85,B 0,C 180,E1 -1172.033,E2 -1172.033} C_VEL
LIN {X 0,Y 594.259,Z 630.318,A -85,B 0,C 180,E1 -1173.389,E2 -1173.389} C_VEL
LIN {X 0,Y 594.237,Z 626.201,A -85,B 0,C 180,E1 -1174.748,E2 -1174.748} C_VEL
LIN {X 0,Y 594.279,Z 620.53,A -85,B 0,C 180,E1 -1176.109,E2 -1176.109} C_VEL
LIN {X 0,Y 594.303,Z 614.13,A -85,B 0,C 180,E1 -1177.303,E2 -1177.303} C_VEL
LIN {X 0,Y 594.323,Z 606.175,A -85,B 0,C 180,E1 -1178.5,E2 -1178.5} C_VEL
LIN {X 0,Y 594.367,Z 597.856,A -85,B 0,C 180,E1 -1179.528,E2 -1179.528} C_VEL
LIN {X 0,Y 594.448,Z 587.844,A -85,B 0,C 180,E1 -1180.559,E2 -1180.559} C_VEL
LIN {X 0,Y 594.523,Z 576.571,A -85,B 0,C 180,E1 -1181.512,E2 -1181.512} C_VEL
LIN {X 0,Y 594.582,Z 564.108,A -85,B 0,C 180,E1 -1182.37,E2 -1182.37} C_VEL
LIN {X 0,Y 594.663,Z 551.651,A -85,B 0,C 180,E1 -1183.063,E2 -1183.063} C_VEL
LIN {X 0,Y 594.74,Z 537.73,A -85,B 0,C 180,E1 -1183.67,E2 -1183.67} C_VEL
LIN {X 0,Y 594.817,Z 524.155,A -85,B 0,C 180,E1 -1184.111,E2 -1184.111} C_VEL
LIN {X 0,Y 594.857,Z 509.923,A -85,B 0,C 180,E1 -1184.43,E2 -1184.43} C_VEL
LIN {X 0,Y 594.884,Z 373.342,A -85,B 0,C 180,E1 -1186.125,E2 -1186.125} C_VEL
LIN {X 0,Y 594.559,Z 371.332,A -85,B 0,C 180,E1 -1186.171,E2 -1186.171} C_VEL
LIN {X 0,Y 594.69,Z 347.364,A -85,B 0,C 180,E1 -1189.108,E2 -1189.108} C_VEL
LIN {X 0,Y 594.825,Z 323.904,A -85,B 0,C 180,E1 -1192.032,E2 -1192.032} C_VEL
LIN {X 0,Y 594.928,Z 307.974,A -85,B 0,C 180,E1 -1194.05,E2 -1194.05} C_VEL
LIN {X 0,Y 594.39,Z 305.072,A -85,B 0,C 180,E1 -1194.468,E2 -1194.468} C_VEL
LIN {X 0,Y 594.384,Z 305.071,A -85,B 0,C 180,E1 -1196.699,E2 -1196.699} C_VEL
LIN {X 0,Y 594.379,Z 305.076,A -85,B 0,C 180,E1 -1198.998,E2 -1198.998} C_VEL
LIN {X 0,Y 594.389,Z 305.066,A -85,B 0,C 180,E1 -1201.644,E2 -1201.644} C_VEL
LIN {X 0,Y 594.395,Z 305.069,A -85,B 0,C 180,E1 -1204.578,E2 -1204.578} C_VEL
LIN {X 0,Y 594.383,Z 305.072,A -85,B 0,C 180,E1 -1207.086,E2 -1207.086} C_VEL
LIN {X 0,Y 594.373,Z 305.067,A -85,B 0,C 180,E1 -1209.774,E2 -1209.774} C_VEL
LIN {X 0,Y 594.364,Z 305.072,A -85,B 0,C 180,E1 -1212.375,E2 -1212.375} C_VEL
LIN {X 0,Y 594.359,Z 305.07,A -85,B 0,C 180,E1 -1215.19,E2 -1215.19} C_VEL
LIN {X 0,Y 594.368,Z 305.067,A -85,B 0,C 180,E1 -1217.624,E2 -1217.624} C_VEL
LIN {X 0,Y 594.386,Z 305.071,A -85,B 0,C 180,E1 -1220.32,E2 -1220.32} C_VEL
LIN {X 0,Y 594.378,Z 305.07,A -85,B 0,C 180,E1 -1222.913,E2 -1222.913} C_VEL
LIN {X 0,Y 594.378,Z 305.068,A -85,B 0,C 180,E1 -1225.86,E2 -1225.86} C_VEL
LIN {X 0,Y 594.363,Z 305.073,A -85,B 0,C 180,E1 -1228.649,E2 -1228.649} C_VEL
LIN {X 0,Y 594.376,Z 305.067,A -85,B 0,C 180,E1 -1231.041,E2 -1231.041} C_VEL
LIN {X 0,Y 594.389,Z 305.07,A -85,B 0,C 180,E1 -1233.974,E2 -1233.974} C_VEL
LIN {X 0,Y 594.374,Z 305.075,A -85,B 0,C 180,E1 -1236.295,E2 -1236.295} C_VEL
LIN {X 0,Y 594.394,Z 305.064,A -85,B 0,C 180,E1 -1239.224,E2 -1239.224} C_VEL
LIN {X 0,Y 594.369,Z 305.077,A -85,B 0,C 180,E1 -1242.095,E2 -1242.095} C_VEL
LIN {X 0,Y 594.354,Z 305.076,A -85,B 0,C 180,E1 -1244.219,E2 -1244.219} C_VEL
LIN {X 0,Y 594.364,Z 305.073,A -85,B 0,C 180,E1 -1246.32,E2 -1246.32} C_VEL
LIN {X 0,Y 594.349,Z 305.069,A -85,B 0,C 180,E1 -1249.094,E2 -1249.094} C_VEL
LIN {X 0,Y 594.402,Z 305.073,A -85,B 0,C 180,E1 -1251.843,E2 -1251.843} C_VEL
LIN {X 0,Y 594.356,Z 305.069,A -85,B 0,C 180,E1 -1254.572,E2 -1254.572} C_VEL
LIN {X 0,Y 594.394,Z 305.066,A -85,B 0,C 180,E1 -1257.289,E2 -1257.289} C_VEL
LIN {X 0,Y 594.393,Z 305.069,A -85,B 0,C 180,E1 -1260,E2 -1260} C_VEL
LIN {X 0,Y 594.362,Z 305.068,A -85,B 0,C 180,E1 -1262.711,E2 -1262.711} C_VEL
LIN {X 0,Y 594.37,Z 305.074,A -85,B 0,C 180,E1 -1265.428,E2 -1265.428} C_VEL
LIN {X 0,Y 594.337,Z 305.072,A -85,B 0,C 180,E1 -1268.158,E2 -1268.158} C_VEL
LIN {X 0,Y 594.353,Z 305.073,A -85,B 0,C 180,E1 -1271.061,E2 -1271.061} C_VEL
LIN {X 0,Y 594.318,Z 305.074,A -85,B 0,C 180,E1 -1274.15,E2 -1274.15} C_VEL
LIN {X 0,Y 594.315,Z 305.077,A -85,B 0,C 180,E1 -1275.279,E2 -1275.279} C_VEL
LIN {X 0,Y 593.641,Z 305.161,A -85,B 0,C 180,E1 -1275.844,E2 -1275.844} C_VEL
LIN {X 0,Y 590.775,Z 305.516,A -85,B 0,C 180,E1 -1276.762,E2 -1276.762} C_VEL
LIN {X 0,Y 588.366,Z 305.823,A -85,B 0,C 180,E1 -1277.501,E2 -1277.501} C_VEL
LIN {X 0,Y 587.343,Z 305.944,A -85,B 0,C 180,E1 -1278.071,E2 -1278.071} C_VEL
LIN {X 0,Y 587.266,Z 305.952,A -85,B 0,C 180,E1 -1278.264,E2 -1278.264} C_VEL
LIN {X 0,Y 587.321,Z 305.951,A -85,B 0,C 180,E1 -1281.038,E2 -1281.038} C_VEL
LIN {X 0,Y 587.274,Z 305.951,A -85,B 0,C 180,E1 -1284.009,E2 -1284.009} C_VEL
LIN {X 0,Y 587.32,Z 305.946,A -85,B 0,C 180,E1 -1286.279,E2 -1286.279} C_VEL
LIN {X 0,Y 587.33,Z 305.953,A -85,B 0,C 180,E1 -1289.132,E2 -1289.132} C_VEL
LIN {X 0,Y 587.329,Z 305.945,A -85,B 0,C 180,E1 -1291.835,E2 -1291.835} C_VEL
LIN {X 0,Y 587.328,Z 305.946,A -85,B 0,C 180,E1 -1294.347,E2 -1294.347} C_VEL
LIN {X 0,Y 587.332,Z 305.945,A -85,B 0,C 180,E1 -1297.608,E2 -1297.608} C_VEL
LIN {X 0,Y 587.299,Z 305.949,A -85,B 0,C 180,E1 -1300.255,E2 -1300.255} C_VEL
LIN {X 0,Y 587.306,Z 305.952,A -85,B 0,C 180,E1 -1303.119,E2 -1303.119} C_VEL
LIN {X 0,Y 587.303,Z 305.948,A -85,B 0,C 180,E1 -1306.049,E2 -1306.049} C_VEL
LIN {X 0,Y 587.329,Z 305.952,A -85,B 0,C 180,E1 -1308.925,E2 -1308.925} C_VEL
LIN {X 0,Y 587.327,Z 305.962,A -85,B 0,C 180,E1 -1311.522,E2 -1311.522} C_VEL
LIN {X 0,Y 587.624,Z 311.605,A -85,B 0,C 180,E1 -1312.414,E2 -1312.414} C_VEL
LIN {X 0,Y 587.517,Z 330.504,A -85,B 0,C 180,E1 -1315.331,E2 -1315.331} C_VEL
LIN {X 0,Y 587.488,Z 332.901,A -85,B 0,C 180,E1 -1315.698,E2 -1315.698} C_VEL
LIN {X 0,Y 588.196,Z 338.344,A -85,B 0,C 180,E1 -1315.794,E2 -1315.794} C_VEL
LIN {X 0,Y 587.981,Z 469.673,A -85,B 0,C 180,E1 -1317.437,E2 -1317.437} C_VEL
LIN {X 0,Y 587.925,Z 484.486,A -85,B 0,C 180,E1 -1317.775,E2 -1317.775} C_VEL
LIN {X 0,Y 587.823,Z 497.877,A -85,B 0,C 180,E1 -1318.217,E2 -1318.217} C_VEL
LIN {X 0,Y 587.714,Z 511.292,A -85,B 0,C 180,E1 -1318.807,E2 -1318.807} C_VEL
LIN {X 0,Y 587.638,Z 524.001,A -85,B 0,C 180,E1 -1319.52,E2 -1319.52} C_VEL
LIN {X 0,Y 587.523,Z 535.795,A -85,B 0,C 180,E1 -1320.336,E2 -1320.336} C_VEL
LIN {X 0,Y 587.435,Z 546.518,A -85,B 0,C 180,E1 -1321.236,E2 -1321.236} C_VEL
LIN {X 0,Y 587.361,Z 555.924,A -85,B 0,C 180,E1 -1322.184,E2 -1322.184} C_VEL
LIN {X 0,Y 587.276,Z 565.418,A -85,B 0,C 180,E1 -1323.336,E2 -1323.336} C_VEL
LIN {X 0,Y 587.227,Z 573.11,A -85,B 0,C 180,E1 -1324.479,E2 -1324.479} C_VEL
LIN {X 0,Y 587.19,Z 579.868,A -85,B 0,C 180,E1 -1325.72,E2 -1325.72} C_VEL
LIN {X 0,Y 587.189,Z 584.336,A -85,B 0,C 180,E1 -1326.737,E2 -1326.737} C_VEL
LIN {X 0,Y 587.168,Z 588.21,A -85,B 0,C 180,E1 -1327.851,E2 -1327.851} C_VEL
LIN {X 0,Y 587.167,Z 591.212,A -85,B 0,C 180,E1 -1329.003,E2 -1329.003} C_VEL
LIN {X 0,Y 587.113,Z 593.542,A -85,B 0,C 180,E1 -1330.418,E2 -1330.418} C_VEL
LIN {X 0,Y 587.125,Z 594.466,A -85,B 0,C 180,E1 -1331.868,E2 -1331.868} C_VEL
LIN {X 0,Y 587.16,Z 593.938,A -85,B 0,C 180,E1 -1333.306,E2 -1333.306} C_VEL
LIN {X 0,Y 587.141,Z 591.95,A -85,B 0,C 180,E1 -1334.733,E2 -1334.733} C_VEL
LIN {X 0,Y 587.179,Z 588.481,A -85,B 0,C 180,E1 -1336.151,E2 -1336.151} C_VEL
LIN {X 0,Y 587.197,Z 583.485,A -85,B 0,C 180,E1 -1337.56,E2 -1337.56} C_VEL
LIN {X 0,Y 587.227,Z 577.016,A -85,B 0,C 180,E1 -1338.926,E2 -1338.926} C_VEL
LIN {X 0,Y 587.28,Z 569.451,A -85,B 0,C 180,E1 -1340.182,E2 -1340.182} C_VEL
LIN {X 0,Y 587.3,Z 560.345,A -85,B 0,C 180,E1 -1341.398,E2 -1341.398} C_VEL
LIN {X 0,Y 587.411,Z 550.835,A -85,B 0,C 180,E1 -1342.438,E2 -1342.438} C_VEL
LIN {X 0,Y 587.48,Z 539.977,A -85,B 0,C 180,E1 -1343.422,E2 -1343.422} C_VEL
LIN {X 0,Y 587.573,Z 528.899,A -85,B 0,C 180,E1 -1344.251,E2 -1344.251} C_VEL
LIN {X 0,Y 587.664,Z 516.219,A -85,B 0,C 180,E1 -1345.027,E2 -1345.027} C_VEL
LIN {X 0,Y 587.788,Z 503.864,A -85,B 0,C 180,E1 -1345.629,E2 -1345.629} C_VEL
LIN {X 0,Y 587.863,Z 490.215,A -85,B 0,C 180,E1 -1346.145,E2 -1346.145} C_VEL
LIN {X 0,Y 587.962,Z 475.902,A -85,B 0,C 180,E1 -1346.531,E2 -1346.531} C_VEL
LIN {X 0,Y 588.018,Z 461.855,A -85,B 0,C 180,E1 -1346.768,E2 -1346.768} C_VEL
LIN {X 0,Y 588.138,Z 336.475,A -85,B 0,C 180,E1 -1348.321,E2 -1348.321} C_VEL
LIN {X 0,Y 587.458,Z 332.897,A -85,B 0,C 180,E1 -1348.394,E2 -1348.394} C_VEL
LIN {X 0,Y 587.611,Z 314.665,A -85,B 0,C 180,E1 -1351.2,E2 -1351.2} C_VEL
LIN {X 0,Y 587.509,Z 306.993,A -85,B 0,C 180,E1 -1352.4,E2 -1352.4} C_VEL
LIN {X 0,Y 587.355,Z 305.946,A -85,B 0,C 180,E1 -1352.572,E2 -1352.572} C_VEL
LIN {X 0,Y 587.352,Z 305.951,A -85,B 0,C 180,E1 -1355.494,E2 -1355.494} C_VEL
LIN {X 0,Y 587.315,Z 305.947,A -85,B 0,C 180,E1 -1358.257,E2 -1358.257} C_VEL
LIN {X 0,Y 587.347,Z 305.95,A -85,B 0,C 180,E1 -1361.134,E2 -1361.134} C_VEL
LIN {X 0,Y 587.329,Z 305.946,A -85,B 0,C 180,E1 -1363.847,E2 -1363.847} C_VEL
LIN {X 0,Y 587.329,Z 305.948,A -85,B 0,C 180,E1 -1366.809,E2 -1366.809} C_VEL
LIN {X 0,Y 587.299,Z 305.951,A -85,B 0,C 180,E1 -1369.577,E2 -1369.577} C_VEL
LIN {X 0,Y 587.3,Z 305.949,A -85,B 0,C 180,E1 -1371.776,E2 -1371.776} C_VEL
LIN {X 0,Y 587.294,Z 305.953,A -85,B 0,C 180,E1 -1374.762,E2 -1374.762} C_VEL
LIN {X 0,Y 587.295,Z 305.949,A -85,B 0,C 180,E1 -1377.683,E2 -1377.683} C_VEL
LIN {X 0,Y 587.29,Z 305.949,A -85,B 0,C 180,E1 -1380.173,E2 -1380.173} C_VEL
LIN {X 0,Y 587.307,Z 305.951,A -85,B 0,C 180,E1 -1382.581,E2 -1382.581} C_VEL
LIN {X 0,Y 587.302,Z 305.955,A -85,B 0,C 180,E1 -1385.058,E2 -1385.058} C_VEL
LIN {X 0,Y 587.277,Z 305.95,A -85,B 0,C 180,E1 -1387.831,E2 -1387.831} C_VEL
LIN {X 0,Y 587.294,Z 305.95,A -85,B 0,C 180,E1 -1390.256,E2 -1390.256} C_VEL
LIN {X 0,Y 587.27,Z 305.956,A -85,B 0,C 180,E1 -1393.114,E2 -1393.114} C_VEL
LIN {X 0,Y 587.284,Z 305.951,A -85,B 0,C 180,E1 -1396.046,E2 -1396.046} C_VEL
LIN {X 0,Y 587.304,Z 305.953,A -85,B 0,C 180,E1 -1398.929,E2 -1398.929} C_VEL
LIN {X 0,Y 587.268,Z 305.952,A -85,B 0,C 180,E1 -1401.516,E2 -1401.516} C_VEL
LIN {X 0,Y 587.267,Z 305.954,A -85,B 0,C 180,E1 -1404.099,E2 -1404.099} C_VEL
LIN {X 0,Y 587.33,Z 305.948,A -85,B 0,C 180,E1 -1406.89,E2 -1406.89} C_VEL
LIN {X 0,Y 587.287,Z 305.949,A -85,B 0,C 180,E1 -1409.499,E2 -1409.499} C_VEL
LIN {X 0,Y 587.295,Z 305.956,A -85,B 0,C 180,E1 -1412.318,E2 -1412.318} C_VEL
LIN {X 0,Y 587.3,Z 305.948,A -85,B 0,C 180,E1 -1415.239,E2 -1415.239} C_VEL
LIN {X 0,Y 587.299,Z 305.956,A -85,B 0,C 180,E1 -1418.225,E2 -1418.225} C_VEL
LIN {X 0,Y 587.324,Z 305.945,A -85,B 0,C 180,E1 -1421.151,E2 -1421.151} C_VEL
LIN {X 0,Y 587.294,Z 305.954,A -85,B 0,C 180,E1 -1424.024,E2 -1424.024} C_VEL
LIN {X 0,Y 587.341,Z 305.952,A -85,B 0,C 180,E1 -1426.154,E2 -1426.154} C_VEL
LIN {X 0,Y 587.339,Z 305.943,A -85,B 0,C 180,E1 -1428.963,E2 -1428.963} C_VEL
LIN {X 0,Y 587.336,Z 305.947,A -85,B 0,C 180,E1 -1431.745,E2 -1431.745} C_VEL
LIN {X 0,Y 587.352,Z 305.945,A -85,B 0,C 180,E1 -1434.507,E2 -1434.507} C_VEL
LIN {X 0,Y 587.351,Z 305.942,A -85,B 0,C 180,E1 -1437.257,E2 -1437.257} C_VEL
LIN {X 0,Y 587.384,Z 305.948,A -85,B 0,C 180,E1 -1440,E2 -1440} C_VEL
LIN {X 0,Y 587.366,Z 305.94,A -85,B 0,C 180,E1 -1442.744,E2 -1442.744} C_VEL
LIN {X 0,Y 587.344,Z 305.946,A -85,B 0,C 180,E1 -1445.493,E2 -1445.493} C_VEL
LIN {X 0,Y 587.365,Z 305.943,A -85,B 0,C 180,E1 -1448.255,E2 -1448.255} C_VEL
LIN {X 0,Y 587.352,Z 305.942,A -85,B 0,C 180,E1 -1451.134,E2 -1451.134} C_VEL
LIN {X 0,Y 587.368,Z 305.942,A -85,B 0,C 180,E1 -1454.26,E2 -1454.26} C_VEL
LIN {X 0,Y 587.343,Z 305.947,A -85,B 0,C 180,E1 -1457.406,E2 -1457.406} C_VEL
LIN {X 0,Y 587.342,Z 305.951,A -85,B 0,C 180,E1 -1459.575,E2 -1459.575} C_VEL
LIN {X 0,Y 587.341,Z 305.942,A -85,B 0,C 180,E1 -1462.514,E2 -1462.514} C_VEL
LIN {X 0,Y 587.338,Z 305.952,A -85,B 0,C 180,E1 -1465.517,E2 -1465.517} C_VEL
LIN {X 0,Y 587.343,Z 305.947,A -85,B 0,C 180,E1 -1467.818,E2 -1467.818} C_VEL
LIN {X 0,Y 587.338,Z 305.943,A -85,B 0,C 180,E1 -1470.509,E2 -1470.509} C_VEL
LIN {X 0,Y 587.338,Z 305.953,A -85,B 0,C 180,E1 -1473.397,E2 -1473.397} C_VEL
LIN {X 0,Y 587.293,Z 305.951,A -85,B 0,C 180,E1 -1475.9,E2 -1475.9} C_VEL
LIN {X 0,Y 587.325,Z 305.944,A -85,B 0,C 180,E1 -1478.48,E2 -1478.48} C_VEL
LIN {X 0,Y 587.339,Z 305.95,A -85,B 0,C 180,E1 -1481.157,E2 -1481.157} C_VEL
LIN {X 0,Y 587.331,Z 305.944,A -85,B 0,C 180,E1 -1484.113,E2 -1484.113} C_VEL
LIN {X 0,Y 587.315,Z 305.952,A -85,B 0,C 180,E1 -1486.993,E2 -1486.993} C_VEL
LIN {X 0,Y 587.319,Z 305.947,A -85,B 0,C 180,E1 -1489.746,E2 -1489.746} C_VEL
LIN {X 0,Y 587.347,Z 305.942,A -85,B 0,C 180,E1 -1492.392,E2 -1492.392} C_VEL
LIN {X 0,Y 587.363,Z 305.94,A -85,B 0,C 180,E1 -1495.78,E2 -1495.78} C_VEL
LIN {X 0,Y 587.34,Z 305.944,A -85,B 0,C 180,E1 -1498.231,E2 -1498.231} C_VEL
LIN {X 0,Y 587.351,Z 305.951,A -85,B 0,C 180,E1 -1500.867,E2 -1500.867} C_VEL
LIN {X 0,Y 587.362,Z 305.942,A -85,B 0,C 180,E1 -1503.819,E2 -1503.819} C_VEL
LIN {X 0,Y 587.366,Z 306.045,A -85,B 0,C 180,E1 -1505.369,E2 -1505.369} C_VEL
LIN {X 0,Y 588.096,Z 310.86,A -85,B 0,C 180,E1 -1506.026,E2 -1506.026} C_VEL
LIN {X 0,Y 587.861,Z 334.031,A -85,B 0,C 180,E1 -1508.982,E2 -1508.982} C_VEL
LIN {X 0,Y 587.714,Z 355.754,A -85,B 0,C 180,E1 -1511.705,E2 -1511.705} C_VEL
LIN {X 0,Y 587.6,Z 371.412,A -85,B 0,C 180,E1 -1513.642,E2 -1513.642} C_VEL
LIN {X 0,Y 588.204,Z 375.574,A -85,B 0,C 180,E1 -1513.715,E2 -1513.715} C_VEL
LIN {X 0,Y 587.995,Z 509.858,A -85,B 0,C 180,E1 -1515.396,E2 -1515.396} C_VEL
LIN {X 0,Y 587.93,Z 524.242,A -85,B 0,C 180,E1 -1515.723,E2 -1515.723} C_VEL
LIN {X 0,Y 587.829,Z 538.824,A -85,B 0,C 180,E1 -1516.209,E2 -1516.209} C_VEL
LIN {X 0,Y 587.728,Z 551.628,A -85,B 0,C 180,E1 -1516.779,E2 -1516.779} C_VEL
LIN {X 0,Y 587.606,Z 564.088,A -85,B 0,C 180,E1 -1517.479,E2 -1517.479} C_VEL
LIN {X 0,Y 587.514,Z 575.469,A -85,B 0,C 180,E1 -1518.266,E2 -1518.266} C_VEL
LIN {X 0,Y 587.467,Z 585.928,A -85,B 0,C 180,E1 -1519.139,E2 -1519.139} C_VEL
LIN {X 0,Y 587.353,Z 596.329,A -85,B 0,C 180,E1 -1520.182,E2 -1520.182} C_VEL
LIN {X 0,Y 587.311,Z 604.908,A -85,B 0,C 180,E1 -1521.223,E2 -1521.223} C_VEL
LIN {X 0,Y 587.249,Z 613.112,A -85,B 0,C 180,E1 -1522.435,E2 -1522.435} C_VEL
LIN {X 0,Y 587.179,Z 619.682,A -85,B 0,C 180,E1 -1523.635,E2 -1523.635} C_VEL
LIN {X 0,Y 587.16,Z 624.959,A -85,B 0,C 180,E1 -1524.849,E2 -1524.849} C_VEL
LIN {X 0,Y 587.179,Z 628.44,A -85,B 0,C 180,E1 -1525.881,E2 -1525.881} C_VEL
LIN {X 0,Y 587.13,Z 631.83,A -85,B 0,C 180,E1 -1527.255,E2 -1527.255} C_VEL
LIN {X 0,Y 587.141,Z 633.831,A -85,B 0,C 180,E1 -1528.628,E2 -1528.628} C_VEL
LIN {X 0,Y 587.135,Z 634.5,A -85,B 0,C 180,E1 -1529.999,E2 -1529.999} C_VEL
LIN {X 0,Y 587.141,Z 633.833,A -85,B 0,C 180,E1 -1531.371,E2 -1531.371} C_VEL
LIN {X 0,Y 587.13,Z 631.834,A -85,B 0,C 180,E1 -1532.744,E2 -1532.744} C_VEL
LIN {X 0,Y 587.179,Z 628.445,A -85,B 0,C 180,E1 -1534.118,E2 -1534.118} C_VEL
LIN {X 0,Y 587.199,Z 623.57,A -85,B 0,C 180,E1 -1535.494,E2 -1535.494} C_VEL
LIN {X 0,Y 587.208,Z 617.056,A -85,B 0,C 180,E1 -1536.873,E2 -1536.873} C_VEL
LIN {X 0,Y 587.268,Z 609.804,A -85,B 0,C 180,E1 -1538.083,E2 -1538.083} C_VEL
LIN {X 0,Y 587.33,Z 600.828,A -85,B 0,C 180,E1 -1539.296,E2 -1539.296} C_VEL
LIN {X 0,Y 587.371,Z 591.398,A -85,B 0,C 180,E1 -1540.339,E2 -1540.339} C_VEL
LIN {X 0,Y 587.474,Z 581.034,A -85,B 0,C 180,E1 -1541.29,E2 -1541.29} C_VEL
LIN {X 0,Y 587.574,Z 569.441,A -85,B 0,C 180,E1 -1542.169,E2 -1542.169} C_VEL
LIN {X 0,Y 587.667,Z 556.661,A -85,B 0,C 180,E1 -1542.957,E2 -1542.957} C_VEL
LIN {X 0,Y 587.78,Z 544.176,A -85,B 0,C 180,E1 -1543.57,E2 -1543.57} C_VEL
LIN {X 0,Y 587.89,Z 530.628,A -85,B 0,C 180,E1 -1544.085,E2 -1544.085} C_VEL
LIN {X 0,Y 587.946,Z 516.986,A -85,B 0,C 180,E1 -1544.461,E2 -1544.461} C_VEL
LIN {X 0,Y 588.008,Z 502.658,A -85,B 0,C 180,E1 -1544.713,E2 -1544.713} C_VEL
LIN {X 0,Y 588.072,Z 374.112,A -85,B 0,C 180,E1 -1546.307,E2 -1546.307} C_VEL
LIN {X 0,Y 587.588,Z 371.332,A -85,B 0,C 180,E1 -1546.368,E2 -1546.368} C_VEL
LIN {X 0,Y 587.748,Z 348.872,A -85,B 0,C 180,E1 -1549.153,E2 -1549.153} C_VEL
LIN {X 0,Y 587.915,Z 326.8,A -85,B 0,C 180,E1 -1551.935,E2 -1551.935} C_VEL
LIN {X 0,Y 588.077,Z 309.589,A -85,B 0,C 180,E1 -1554.139,E2 -1554.139} C_VEL
LIN {X 0,Y 587.36,Z 305.947,A -85,B 0,C 180,E1 -1554.661,E2 -1554.661} C_VEL
LIN {X 0,Y 587.329,Z 305.954,A -85,B 0,C 180,E1 -1557.045,E2 -1557.045} C_VEL
LIN {X 0,Y 587.346,Z 305.947,A -85,B 0,C 180,E1 -1559.379,E2 -1559.379} C_VEL
LIN {X 0,Y 587.351,Z 305.942,A -85,B 0,C 180,E1 -1561.836,E2 -1561.836} C_VEL
LIN {X 0,Y 587.353,Z 305.943,A -85,B 0,C 180,E1 -1564.348,E2 -1564.348} C_VEL
LIN {X 0,Y 587.35,Z 305.95,A -85,B 0,C 180,E1 -1566.746,E2 -1566.746} C_VEL
LIN {X 0,Y 587.343,Z 305.944,A -85,B 0,C 180,E1 -1569.358,E2 -1569.358} C_VEL
LIN {X 0,Y 587.33,Z 305.945,A -85,B 0,C 180,E1 -1572.107,E2 -1572.107} C_VEL
LIN {X 0,Y 587.311,Z 305.949,A -85,B 0,C 180,E1 -1575.088,E2 -1575.088} C_VEL
LIN {X 0,Y 587.348,Z 305.943,A -85,B 0,C 180,E1 -1577.927,E2 -1577.927} C_VEL
LIN {X 0,Y 587.327,Z 305.946,A -85,B 0,C 180,E1 -1581.057,E2 -1581.057} C_VEL
LIN {X 0,Y 587.347,Z 305.942,A -85,B 0,C 180,E1 -1583.291,E2 -1583.291} C_VEL
LIN {X 0,Y 587.356,Z 305.942,A -85,B 0,C 180,E1 -1585.779,E2 -1585.779} C_VEL
LIN {X 0,Y 587.338,Z 305.95,A -85,B 0,C 180,E1 -1588.231,E2 -1588.231} C_VEL
LIN {X 0,Y 587.344,Z 305.944,A -85,B 0,C 180,E1 -1590.866,E2 -1590.866} C_VEL
LIN {X 0,Y 587.357,Z 305.943,A -85,B 0,C 180,E1 -1593.817,E2 -1593.817} C_VEL
LIN {X 0,Y 587.325,Z 305.951,A -85,B 0,C 180,E1 -1595.993,E2 -1595.993} C_VEL
LIN {X 0,Y 587.312,Z 305.956,A -85,B 0,C 180,E1 -1598.225,E2 -1598.225} C_VEL
LIN {X 0,Y 587.338,Z 305.942,A -85,B 0,C 180,E1 -1601.151,E2 -1601.151} C_VEL
LIN {X 0,Y 587.312,Z 305.956,A -85,B 0,C 180,E1 -1604.024,E2 -1604.024} C_VEL
LIN {X 0,Y 587.345,Z 305.95,A -85,B 0,C 180,E1 -1606.154,E2 -1606.154} C_VEL
LIN {X 0,Y 587.327,Z 305.943,A -85,B 0,C 180,E1 -1608.962,E2 -1608.962} C_VEL
LIN {X 0,Y 587.354,Z 305.949,A -85,B 0,C 180,E1 -1611.744,E2 -1611.744} C_VEL
LIN {X 0,Y 587.325,Z 305.946,A -85,B 0,C 180,E1 -1614.506,E2 -1614.506} C_VEL
LIN {X 0,Y 587.357,Z 305.942,A -85,B 0,C 180,E1 -1617.256,E2 -1617.256} C_VEL
LIN {X 0,Y 587.362,Z 305.945,A -85,B 0,C 180,E1 -1620,E2 -1620} C_VEL
LIN {X 0,Y 587.332,Z 305.944,A -85,B 0,C 180,E1 -1622.743,E2 -1622.743} C_VEL
LIN {X 0,Y 587.334,Z 305.951,A -85,B 0,C 180,E1 -1625.493,E2 -1625.493} C_VEL
LIN {X 0,Y 587.303,Z 305.948,A -85,B 0,C 180,E1 -1628.256,E2 -1628.256} C_VEL
LIN {X 0,Y 587.32,Z 305.95,A -85,B 0,C 180,E1 -1631.124,E2 -1631.124} C_VEL
LIN {X 0,Y 587.289,Z 305.949,A -85,B 0,C 180,E1 -1634.235,E2 -1634.235} C_VEL
LIN {X 0,Y 587.304,Z 305.949,A -85,B 0,C 180,E1 -1636.803,E2 -1636.803} C_VEL
LIN {X 0,Y 587.266,Z 305.952,A -85,B 0,C 180,E1 -1638.264,E2 -1638.264} C_VEL
LIN {X 0,Y 586.631,Z 306.035,A -85,B 0,C 180,E1 -1638.836,E2 -1638.836} C_VEL
LIN {X 0,Y 583.834,Z 306.383,A -85,B 0,C 180,E1 -1639.765,E2 -1639.765} C_VEL
LIN {X 0,Y 581.437,Z 306.683,A -85,B 0,C 180,E1 -1640.512,E2 -1640.512} C_VEL
LIN {X 0,Y 580.376,Z 306.818,A -85,B 0,C 180,E1 -1641.088,E2 -1641.088} C_VEL
LIN {X 0,Y 580.274,Z 306.832,A -85,B 0,C 180,E1 -1641.283,E2 -1641.283} C_VEL
LIN {X 0,Y 580.238,Z 306.832,A -85,B 0,C 180,E1 -1643.559,E2 -1643.559} C_VEL
LIN {X 0,Y 580.274,Z 306.824,A -85,B 0,C 180,E1 -1646.333,E2 -1646.333} C_VEL
LIN {X 0,Y 580.263,Z 306.832,A -85,B 0,C 180,E1 -1649.305,E2 -1649.305} C_VEL
LIN {X 0,Y 580.283,Z 306.822,A -85,B 0,C 180,E1 -1652.201,E2 -1652.201} C_VEL
LIN {X 0,Y 580.275,Z 306.829,A -85,B 0,C 180,E1 -1654.697,E2 -1654.697} C_VEL
LIN {X 0,Y 580.287,Z 306.827,A -85,B 0,C 180,E1 -1657.269,E2 -1657.269} C_VEL
LIN {X 0,Y 580.279,Z 306.824,A -85,B 0,C 180,E1 -1660.27,E2 -1660.27} C_VEL
LIN {X 0,Y 580.268,Z 306.832,A -85,B 0,C 180,E1 -1662.707,E2 -1662.707} C_VEL
LIN {X 0,Y 580.246,Z 306.827,A -85,B 0,C 180,E1 -1665.611,E2 -1665.611} C_VEL
LIN {X 0,Y 580.269,Z 306.828,A -85,B 0,C 180,E1 -1668.232,E2 -1668.232} C_VEL
LIN {X 0,Y 580.293,Z 306.828,A -85,B 0,C 180,E1 -1671.191,E2 -1671.191} C_VEL
LIN {X 0,Y 580.32,Z 306.924,A -85,B 0,C 180,E1 -1671.415,E2 -1671.415} C_VEL
LIN {X 0,Y 580.647,Z 311.188,A -85,B 0,C 180,E1 -1672.103,E2 -1672.103} C_VEL
LIN {X 0,Y 580.528,Z 330.413,A -85,B 0,C 180,E1 -1675.11,E2 -1675.11} C_VEL
LIN {X 0,Y 580.526,Z 333.143,A -85,B 0,C 180,E1 -1675.508,E2 -1675.508} C_VEL
LIN {X 0,Y 581.384,Z 338.634,A -85,B 0,C 180,E1 -1675.602,E2 -1675.602} C_VEL
LIN {X 0,Y 581.127,Z 469.701,A -85,B 0,C 180,E1 -1677.262,E2 -1677.262} C_VEL
LIN {X 0,Y 581.043,Z 484.093,A -85,B 0,C 180,E1 -1677.591,E2 -1677.591} C_VEL
LIN {X 0,Y 580.925,Z 497.732,A -85,B 0,C 180,E1 -1678.044,E2 -1678.044} C_VEL
LIN {X 0,Y 580.79,Z 511.3,A -85,B 0,C 180,E1 -1678.646,E2 -1678.646} C_VEL
LIN {X 0,Y 580.674,Z 524.279,A -85,B 0,C 180,E1 -1679.384,E2 -1679.384} C_VEL
LIN {X 0,Y 580.541,Z 536.448,A -85,B 0,C 180,E1 -1680.243,E2 -1680.243} C_VEL
LIN {X 0,Y 580.422,Z 547.859,A -85,B 0,C 180,E1 -1681.23,E2 -1681.23} C_VEL
LIN {X 0,Y 580.289,Z 558.562,A -85,B 0,C 180,E1 -1682.367,E2 -1682.367} C_VEL
LIN {X 0,Y 580.204,Z 567.753,A -85,B 0,C 180,E1 -1683.561,E2 -1683.561} C_VEL
LIN {X 0,Y 580.146,Z 575.049,A -85,B 0,C 180,E1 -1684.722,E2 -1684.722} C_VEL
LIN {X 0,Y 580.127,Z 581.782,A -85,B 0,C 180,E1 -1686.057,E2 -1686.057} C_VEL
LIN {X 0,Y 580.073,Z 586.233,A -85,B 0,C 180,E1 -1687.189,E2 -1687.189} C_VEL
LIN {X 0,Y 580.068,Z 588.638,A -85,B 0,C 180,E1 -1687.94,E2 -1687.94} C_VEL
LIN {X 0,Y 580.063,Z 591.063,A -85,B 0,C 180,E1 -1688.895,E2 -1688.895} C_VEL
LIN {X 0,Y 580.018,Z 593.281,A -85,B 0,C 180,E1 -1690.168,E2 -1690.168} C_VEL
LIN {X 0,Y 580.034,Z 594.415,A -85,B 0,C 180,E1 -1691.638,E2 -1691.638} C_VEL
LIN {X 0,Y 580.032,Z 594.095,A -85,B 0,C 180,E1 -1693.095,E2 -1693.095} C_VEL
LIN {X 0,Y 580.037,Z 592.343,A -85,B 0,C 180,E1 -1694.541,E2 -1694.541} C_VEL
LIN {X 0,Y 580.08,Z 589.14,A -85,B 0,C 180,E1 -1695.978,E2 -1695.978} C_VEL
LIN {X 0,Y 580.106,Z 584.391,A -85,B 0,C 180,E1 -1697.405,E2 -1697.405} C_VEL
LIN {X 0,Y 580.11,Z 579.764,A -85,B 0,C 180,E1 -1698.47,E2 -1698.47} C_VEL
LIN {X 0,Y 580.154,Z 573.086,A -85,B 0,C 180,E1 -1699.708,E2 -1699.708} C_VEL
LIN {X 0,Y 580.269,Z 564.809,A -85,B 0,C 180,E1 -1700.942,E2 -1700.942} C_VEL
LIN {X 0,Y 580.337,Z 556.214,A -85,B 0,C 180,E1 -1701.995,E2 -1701.995} C_VEL
LIN {X 0,Y 580.419,Z 545.86,A -85,B 0,C 180,E1 -1703.046,E2 -1703.046} C_VEL
LIN {X 0,Y 580.55,Z 534.349,A -85,B 0,C 180,E1 -1704.007,E2 -1704.007} C_VEL
LIN {X 0,Y 580.67,Z 522.899,A -85,B 0,C 180,E1 -1704.793,E2 -1704.793} C_VEL
LIN {X 0,Y 580.823,Z 510.371,A -85,B 0,C 180,E1 -1705.49,E2 -1705.49} C_VEL
LIN {X 0,Y 580.933,Z 497.502,A -85,B 0,C 180,E1 -1706.055,E2 -1706.055} C_VEL
LIN {X 0,Y 581.036,Z 483.688,A -85,B 0,C 180,E1 -1706.512,E2 -1706.512} C_VEL
LIN {X 0,Y 581.141,Z 469.179,A -85,B 0,C 180,E1 -1706.838,E2 -1706.838} C_VEL
LIN {X 0,Y 581.316,Z 337.299,A -85,B 0,C 180,E1 -1708.507,E2 -1708.507} C_VEL
LIN {X 0,Y 580.459,Z 332.931,A -85,B 0,C 180,E1 -1708.591,E2 -1708.591} C_VEL
LIN {X 0,Y 580.662,Z 314.986,A -85,B 0,C 180,E1 -1711.388,E2 -1711.388} C_VEL
LIN {X 0,Y 580.576,Z 308.414,A -85,B 0,C 180,E1 -1712.429,E2 -1712.429} C_VEL
LIN {X 0,Y 580.314,Z 306.825,A -85,B 0,C 180,E1 -1712.712,E2 -1712.712} C_VEL
LIN {X 0,Y 580.315,Z 306.827,A -85,B 0,C 180,E1 -1715.56,E2 -1715.56} C_VEL
LIN {X 0,Y 580.29,Z 306.822,A -85,B 0,C 180,E1 -1718.357,E2 -1718.357} C_VEL
LIN {X 0,Y 580.299,Z 306.829,A -85,B 0,C 180,E1 -1721.192,E2 -1721.192} C_VEL
LIN {X 0,Y 580.285,Z 306.822,A -85,B 0,C 180,E1 -1724.018,E2 -1724.018} C_VEL
LIN {X 0,Y 580.289,Z 306.826,A -85,B 0,C 180,E1 -1726.907,E2 -1726.907} C_VEL
LIN {X 0,Y 580.274,Z 306.824,A -85,B 0,C 180,E1 -1729.824,E2 -1729.824} C_VEL
LIN {X 0,Y 580.245,Z 306.826,A -85,B 0,C 180,E1 -1732.054,E2 -1732.054} C_VEL
LIN {X 0,Y 580.27,Z 306.834,A -85,B 0,C 180,E1 -1735.082,E2 -1735.082} C_VEL
LIN {X 0,Y 580.242,Z 306.827,A -85,B 0,C 180,E1 -1737.849,E2 -1737.849} C_VEL
LIN {X 0,Y 580.254,Z 306.83,A -85,B 0,C 180,E1 -1740.69,E2 -1740.69} C_VEL
LIN {X 0,Y 580.241,Z 306.831,A -85,B 0,C 180,E1 -1743.307,E2 -1743.307} C_VEL
LIN {X 0,Y 580.217,Z 306.83,A -85,B 0,C 180,E1 -1745.753,E2 -1745.753} C_VEL
LIN {X 0,Y 580.237,Z 306.828,A -85,B 0,C 180,E1 -1748.151,E2 -1748.151} C_VEL
LIN {X 0,Y 580.266,Z 306.834,A -85,B 0,C 180,E1 -1750.847,E2 -1750.847} C_VEL
LIN {X 0,Y 580.209,Z 306.831,A -85,B 0,C 180,E1 -1753.665,E2 -1753.665} C_VEL
LIN {X 0,Y 580.222,Z 306.838,A -85,B 0,C 180,E1 -1756.615,E2 -1756.615} C_VEL
LIN {X 0,Y 580.25,Z 306.829,A -85,B 0,C 180,E1 -1759.153,E2 -1759.153} C_VEL
LIN {X 0,Y 580.235,Z 306.828,A -85,B 0,C 180,E1 -1761.934,E2 -1761.934} C_VEL
LIN {X 0,Y 580.216,Z 306.838,A -85,B 0,C 180,E1 -1764.451,E2 -1764.451} C_VEL
LIN {X 0,Y 580.28,Z 306.825,A -85,B 0,C 180,E1 -1766.975,E2 -1766.975} C_VEL
LIN {X 0,Y 580.252,Z 306.825,A -85,B 0,C 180,E1 -1769.423,E2 -1769.423} C_VEL
LIN {X 0,Y 580.239,Z 306.832,A -85,B 0,C 180,E1 -1772.153,E2 -1772.153} C_VEL
LIN {X 0,Y 580.279,Z 306.825,A -85,B 0,C 180,E1 -1774.919,E2 -1774.919} C_VEL
LIN {X 0,Y 580.233,Z 306.831,A -85,B 0,C 180,E1 -1777.946,E2 -1777.946} C_VEL
LIN {X 0,Y 580.28,Z 306.824,A -85,B 0,C 180,E1 -1780.913,E2 -1780.913} C_VEL
LIN {X 0,Y 580.24,Z 306.83,A -85,B 0,C 180,E1 -1783.825,E2 -1783.825} C_VEL
LIN {X 0,Y 580.297,Z 306.826,A -85,B 0,C 180,E1 -1785.983,E2 -1785.983} C_VEL
LIN {X 0,Y 580.308,Z 306.82,A -85,B 0,C 180,E1 -1788.827,E2 -1788.827} C_VEL
LIN {X 0,Y 580.305,Z 306.822,A -85,B 0,C 180,E1 -1791.644,E2 -1791.644} C_VEL
LIN {X 0,Y 580.318,Z 306.822,A -85,B 0,C 180,E1 -1794.44,E2 -1794.44} C_VEL
LIN {X 0,Y 580.32,Z 306.817,A -85,B 0,C 180,E1 -1797.224,E2 -1797.224} C_VEL
LIN {X 0,Y 580.353,Z 306.823,A -85,B 0,C 180,E1 -1800,E2 -1800} C_VEL
LIN {X 0,Y 580.331,Z 306.816,A -85,B 0,C 180,E1 -1802.777,E2 -1802.777} C_VEL
LIN {X 0,Y 580.313,Z 306.823,A -85,B 0,C 180,E1 -1805.56,E2 -1805.56} C_VEL
LIN {X 0,Y 580.328,Z 306.819,A -85,B 0,C 180,E1 -1808.356,E2 -1808.356} C_VEL
LIN {X 0,Y 580.304,Z 306.821,A -85,B 0,C 180,E1 -1811.191,E2 -1811.191} C_VEL
LIN {X 0,Y 580.326,Z 306.822,A -85,B 0,C 180,E1 -1814.017,E2 -1814.017} C_VEL
LIN {X 0,Y 580.316,Z 306.818,A -85,B 0,C 180,E1 -1816.914,E2 -1816.914} C_VEL
LIN {X 0,Y 580.304,Z 306.826,A -85,B 0,C 180,E1 -1819.823,E2 -1819.823} C_VEL
LIN {X 0,Y 580.292,Z 306.821,A -85,B 0,C 180,E1 -1822.803,E2 -1822.803} C_VEL
LIN {X 0,Y 580.31,Z 306.821,A -85,B 0,C 180,E1 -1825.08,E2 -1825.08} C_VEL
LIN {X 0,Y 580.299,Z 306.821,A -85,B 0,C 180,E1 -1828.186,E2 -1828.186} C_VEL
LIN {X 0,Y 580.285,Z 306.822,A -85,B 0,C 180,E1 -1830.694,E2 -1830.694} C_VEL
LIN {X 0,Y 580.307,Z 306.827,A -85,B 0,C 180,E1 -1833.316,E2 -1833.316} C_VEL
LIN {X 0,Y 580.248,Z 306.83,A -85,B 0,C 180,E1 -1835.756,E2 -1835.756} C_VEL
LIN {X 0,Y 580.289,Z 306.821,A -85,B 0,C 180,E1 -1838.147,E2 -1838.147} C_VEL
LIN {X 0,Y 580.3,Z 306.822,A -85,B 0,C 180,E1 -1840.843,E2 -1840.843} C_VEL
LIN {X 0,Y 580.283,Z 306.825,A -85,B 0,C 180,E1 -1843.658,E2 -1843.658} C_VEL
LIN {X 0,Y 580.276,Z 306.824,A -85,B 0,C 180,E1 -1846.61,E2 -1846.61} C_VEL
LIN {X 0,Y 580.301,Z 306.83,A -85,B 0,C 180,E1 -1849.156,E2 -1849.156} C_VEL
LIN {X 0,Y 580.293,Z 306.821,A -85,B 0,C 180,E1 -1851.927,E2 -1851.927} C_VEL
LIN {X 0,Y 580.256,Z 306.826,A -85,B 0,C 180,E1 -1854.453,E2 -1854.453} C_VEL
LIN {X 0,Y 580.291,Z 306.83,A -85,B 0,C 180,E1 -1856.975,E2 -1856.975} C_VEL
LIN {X 0,Y 580.288,Z 306.826,A -85,B 0,C 180,E1 -1859.424,E2 -1859.424} C_VEL
LIN {X 0,Y 580.299,Z 306.822,A -85,B 0,C 180,E1 -1862.141,E2 -1862.141} C_VEL
LIN {X 0,Y 580.329,Z 306.911,A -85,B 0,C 180,E1 -1865.166,E2 -1865.166} C_VEL
LIN {X 0,Y 581.255,Z 312.308,A -85,B 0,C 180,E1 -1865.916,E2 -1865.916} C_VEL
LIN {X 0,Y 580.969,Z 335.479,A -85,B 0,C 180,E1 -1868.906,E2 -1868.906} C_VEL
LIN {X 0,Y 580.751,Z 358.65,A -85,B 0,C 180,E1 -1871.843,E2 -1871.843} C_VEL
LIN {X 0,Y 580.628,Z 371.412,A -85,B 0,C 180,E1 -1873.44,E2 -1873.44} C_VEL
LIN {X 0,Y 581.397,Z 377.363,A -85,B 0,C 180,E1 -1873.541,E2 -1873.541} C_VEL
LIN {X 0,Y 581.146,Z 509.858,A -85,B 0,C 180,E1 -1875.22,E2 -1875.22} C_VEL
LIN {X 0,Y 581.042,Z 524.476,A -85,B 0,C 180,E1 -1875.557,E2 -1875.557} C_VEL
LIN {X 0,Y 580.92,Z 538.826,A -85,B 0,C 180,E1 -1876.042,E2 -1876.042} C_VEL
LIN {X 0,Y 580.788,Z 551.63,A -85,B 0,C 180,E1 -1876.618,E2 -1876.618} C_VEL
LIN {X 0,Y 580.657,Z 564.09,A -85,B 0,C 180,E1 -1877.327,E2 -1877.327} C_VEL
LIN {X 0,Y 580.527,Z 576.633,A -85,B 0,C 180,E1 -1878.211,E2 -1878.211} C_VEL
LIN {X 0,Y 580.442,Z 587.902,A -85,B 0,C 180,E1 -1879.19,E2 -1879.19} C_VEL
LIN {X 0,Y 580.275,Z 597.846,A -85,B 0,C 180,E1 -1880.237,E2 -1880.237} C_VEL
LIN {X 0,Y 580.241,Z 606.168,A -85,B 0,C 180,E1 -1881.291,E2 -1881.291} C_VEL
LIN {X 0,Y 580.166,Z 614.123,A -85,B 0,C 180,E1 -1882.517,E2 -1882.517} C_VEL
LIN {X 0,Y 580.093,Z 620.525,A -85,B 0,C 180,E1 -1883.74,E2 -1883.74} C_VEL
LIN {X 0,Y 580.078,Z 624.959,A -85,B 0,C 180,E1 -1884.786,E2 -1884.786} C_VEL
LIN {X 0,Y 580.102,Z 628.441,A -85,B 0,C 180,E1 -1885.831,E2 -1885.831} C_VEL
LIN {X 0,Y 580.041,Z 631.83,A -85,B 0,C 180,E1 -1887.221,E2 -1887.221} C_VEL
LIN {X 0,Y 580.041,Z 633.831,A -85,B 0,C 180,E1 -1888.611,E2 -1888.611} C_VEL
LIN {X 0,Y 580.036,Z 634.5,A -85,B 0,C 180,E1 -1889.999,E2 -1889.999} C_VEL
LIN {X 0,Y 580.041,Z 633.833,A -85,B 0,C 180,E1 -1891.388,E2 -1891.388} C_VEL
LIN {X 0,Y 580.041,Z 631.834,A -85,B 0,C 180,E1 -1892.777,E2 -1892.777} C_VEL
LIN {X 0,Y 580.102,Z 628.446,A -85,B 0,C 180,E1 -1894.168,E2 -1894.168} C_VEL
LIN {X 0,Y 580.128,Z 623.571,A -85,B 0,C 180,E1 -1895.561,E2 -1895.561} C_VEL
LIN {X 0,Y 580.14,Z 617.056,A -85,B 0,C 180,E1 -1896.957,E2 -1896.957} C_VEL
LIN {X 0,Y 580.192,Z 609.805,A -85,B 0,C 180,E1 -1898.182,E2 -1898.182} C_VEL
LIN {X 0,Y 580.286,Z 600.828,A -85,B 0,C 180,E1 -1899.41,E2 -1899.41} C_VEL
LIN {X 0,Y 580.356,Z 591.399,A -85,B 0,C 180,E1 -1900.465,E2 -1900.465} C_VEL
LIN {X 0,Y 580.474,Z 581.328,A -85,B 0,C 180,E1 -1901.403,E2 -1901.403} C_VEL
LIN {X 0,Y 580.596,Z 569.443,A -85,B 0,C 180,E1 -1902.318,E2 -1902.318} C_VEL
LIN {X 0,Y 580.731,Z 556.659,A -85,B 0,C 180,E1 -1903.115,E2 -1903.115} C_VEL
LIN {X 0,Y 580.86,Z 544.173,A -85,B 0,C 180,E1 -1903.735,E2 -1903.735} C_VEL
LIN {X 0,Y 581.01,Z 531.199,A -85,B 0,C 180,E1 -1904.235,E2 -1904.235} C_VEL
LIN {X 0,Y 581.082,Z 517.198,A -85,B 0,C 180,E1 -1904.63,E2 -1904.63} C_VEL
LIN {X 0,Y 581.157,Z 502.658,A -85,B 0,C 180,E1 -1904.89,E2 -1904.89} C_VEL
LIN {X 0,Y 581.292,Z 375.23,A -85,B 0,C 180,E1 -1906.489,E2 -1906.489} C_VEL
LIN {X 0,Y 580.634,Z 371.332,A -85,B 0,C 180,E1 -1906.57,E2 -1906.57} C_VEL
LIN {X 0,Y 580.837,Z 348.111,A -85,B 0,C 180,E1 -1909.487,E2 -1909.487} C_VEL
LIN {X 0,Y 581.079,Z 325.352,A -85,B 0,C 180,E1 -1912.394,E2 -1912.394} C_VEL
LIN {X 0,Y 581.175,Z 310.87,A -85,B 0,C 180,E1 -1914.276,E2 -1914.276} C_VEL
LIN {X 0,Y 580.294,Z 306.828,A -85,B 0,C 180,E1 -1914.866,E2 -1914.866} C_VEL
LIN {X 0,Y 580.295,Z 306.822,A -85,B 0,C 180,E1 -1917.858,E2 -1917.858} C_VEL
LIN {X 0,Y 580.29,Z 306.827,A -85,B 0,C 180,E1 -1920.695,E2 -1920.695} C_VEL
LIN {X 0,Y 580.3,Z 306.823,A -85,B 0,C 180,E1 -1923.316,E2 -1923.316} C_VEL
LIN {X 0,Y 580.324,Z 306.817,A -85,B 0,C 180,E1 -1925.767,E2 -1925.767} C_VEL
LIN {X 0,Y 580.286,Z 306.823,A -85,B 0,C 180,E1 -1928.145,E2 -1928.145} C_VEL
LIN {X 0,Y 580.296,Z 306.828,A -85,B 0,C 180,E1 -1930.842,E2 -1930.842} C_VEL
LIN {X 0,Y 580.274,Z 306.823,A -85,B 0,C 180,E1 -1933.657,E2 -1933.657} C_VEL
LIN {X 0,Y 580.281,Z 306.83,A -85,B 0,C 180,E1 -1936.608,E2 -1936.608} C_VEL
LIN {X 0,Y 580.296,Z 306.821,A -85,B 0,C 180,E1 -1939.156,E2 -1939.156} C_VEL
LIN {X 0,Y 580.285,Z 306.823,A -85,B 0,C 180,E1 -1941.926,E2 -1941.926} C_VEL
LIN {X 0,Y 580.281,Z 306.832,A -85,B 0,C 180,E1 -1944.455,E2 -1944.455} C_VEL
LIN {X 0,Y 580.286,Z 306.823,A -85,B 0,C 180,E1 -1946.975,E2 -1946.975} C_VEL
LIN {X 0,Y 580.296,Z 306.82,A -85,B 0,C 180,E1 -1949.425,E2 -1949.425} C_VEL
LIN {X 0,Y 580.313,Z 306.825,A -85,B 0,C 180,E1 -1952.136,E2 -1952.136} C_VEL
LIN {X 0,Y 580.301,Z 306.821,A -85,B 0,C 180,E1 -1954.92,E2 -1954.92} C_VEL
LIN {X 0,Y 580.262,Z 306.83,A -85,B 0,C 180,E1 -1957.947,E2 -1957.947} C_VEL
LIN {X 0,Y 580.29,Z 306.82,A -85,B 0,C 180,E1 -1960.913,E2 -1960.913} C_VEL
LIN {X 0,Y 580.264,Z 306.83,A -85,B 0,C 180,E1 -1963.825,E2 -1963.825} C_VEL
LIN {X 0,Y 580.314,Z 306.827,A -85,B 0,C 180,E1 -1965.983,E2 -1965.983} C_VEL
LIN {X 0,Y 580.296,Z 306.819,A -85,B 0,C 180,E1 -1968.827,E2 -1968.827} C_VEL
LIN {X 0,Y 580.316,Z 306.824,A -85,B 0,C 180,E1 -1971.644,E2 -1971.644} C_VEL
LIN {X 0,Y 580.269,Z 306.831,A -85,B 0,C 180,E1 -1973.742,E2 -1973.742} C_VEL
LIN {X 0,Y 580.255,Z 306.835,A -85,B 0,C 180,E1 -1975.832,E2 -1975.832} C_VEL
LIN {X 0,Y 580.317,Z 306.825,A -85,B 0,C 180,E1 -1977.918,E2 -1977.918} C_VEL
LIN {X 0,Y 580.332,Z 306.821,A -85,B 0,C 180,E1 -1980,E2 -1980} C_VEL
LIN {X 0,Y 580.302,Z 306.82,A -85,B 0,C 180,E1 -1982.776,E2 -1982.776} C_VEL
LIN {X 0,Y 580.298,Z 306.829,A -85,B 0,C 180,E1 -1985.56,E2 -1985.56} C_VEL
LIN {X 0,Y 580.275,Z 306.823,A -85,B 0,C 180,E1 -1988.357,E2 -1988.357} C_VEL
LIN {X 0,Y 580.29,Z 306.826,A -85,B 0,C 180,E1 -1991.191,E2 -1991.191} C_VEL
LIN {X 0,Y 580.255,Z 306.826,A -85,B 0,C 180,E1 -1994.319,E2 -1994.319} C_VEL
LIN {X 0,Y 580.256,Z 306.828,A -85,B 0,C 180,E1 -1996.899,E2 -1996.899} C_VEL
LIN {X 0,Y 580.261,Z 306.827,A -85,B 0,C 180,E1 -1999.824,E2 -1999.824} C_VEL
LIN {X 0,Y 580.274,Z 306.832,A -85,B 0,C 180,E1 -2001.283,E2 -2001.283} C_VEL
LIN {X 0,Y 579.558,Z 306.923,A -85,B 0,C 180,E1 -2001.863,E2 -2001.863} C_VEL
LIN {X 0,Y 576.67,Z 307.279,A -85,B 0,C 180,E1 -2002.803,E2 -2002.803} C_VEL
LIN {X 0,Y 574.27,Z 307.576,A -85,B 0,C 180,E1 -2003.559,E2 -2003.559} C_VEL
LIN {X 0,Y 573.258,Z 307.697,A -85,B 0,C 180,E1 -2004.143,E2 -2004.143} C_VEL
LIN {X 0,Y 573.184,Z 307.706,A -85,B 0,C 180,E1 -2004.34,E2 -2004.34} C_VEL
LIN {X 0,Y 573.2,Z 307.712,A -85,B 0,C 180,E1 -2006.978,E2 -2006.978} C_VEL
LIN {X 0,Y 573.21,Z 307.708,A -85,B 0,C 180,E1 -2009.484,E2 -2009.484} C_VEL
LIN {X 0,Y 573.236,Z 307.7,A -85,B 0,C 180,E1 -2012.228,E2 -2012.228} C_VEL
LIN {X 0,Y 573.222,Z 307.708,A -85,B 0,C 180,E1 -2014.771,E2 -2014.771} C_VEL
LIN {X 0,Y 573.222,Z 307.702,A -85,B 0,C 180,E1 -2017.808,E2 -2017.808} C_VEL
LIN {X 0,Y 573.235,Z 307.704,A -85,B 0,C 180,E1 -2020.526,E2 -2020.526} C_VEL
LIN {X 0,Y 573.228,Z 307.703,A -85,B 0,C 180,E1 -2023.36,E2 -2023.36} C_VEL
LIN {X 0,Y 573.229,Z 307.709,A -85,B 0,C 180,E1 -2026.641,E2 -2026.641} C_VEL
LIN {X 0,Y 573.236,Z 307.703,A -85,B 0,C 180,E1 -2029.475,E2 -2029.475} C_VEL
LIN {X 0,Y 573.285,Z 307.872,A -85,B 0,C 180,E1 -2031.303,E2 -2031.303} C_VEL
LIN {X 0,Y 573.696,Z 311.71,A -85,B 0,C 180,E1 -2031.934,E2 -2031.934} C_VEL
LIN {X 0,Y 573.526,Z 330.025,A -85,B 0,C 180,E1 -2034.836,E2 -2034.836} C_VEL
LIN {X 0,Y 573.514,Z 332.889,A -85,B 0,C 180,E1 -2035.286,E2 -2035.286} C_VEL
LIN {X 0,Y 574.592,Z 339.464,A -85,B 0,C 180,E1 -2035.413,E2 -2035.413} C_VEL
LIN {X 0,Y 574.26,Z 469.738,A -85,B 0,C 180,E1 -2037.082,E2 -2037.082} C_VEL
LIN {X 0,Y 574.148,Z 484.093,A -85,B 0,C 180,E1 -2037.413,E2 -2037.413} C_VEL
LIN {X 0,Y 574.02,Z 497.872,A -85,B 0,C 180,E1 -2037.878,E2 -2037.878} C_VEL
LIN {X 0,Y 573.888,Z 510.314,A -85,B 0,C 180,E1 -2038.432,E2 -2038.432} C_VEL
LIN {X 0,Y 573.698,Z 523.47,A -85,B 0,C 180,E1 -2039.176,E2 -2039.176} C_VEL
LIN {X 0,Y 573.58,Z 535.457,A -85,B 0,C 180,E1 -2040.021,E2 -2040.021} C_VEL
LIN {X 0,Y 573.401,Z 546.26,A -85,B 0,C 180,E1 -2040.945,E2 -2040.945} C_VEL
LIN {X 0,Y 573.295,Z 556.132,A -85,B 0,C 180,E1 -2041.962,E2 -2041.962} C_VEL
LIN {X 0,Y 573.161,Z 565.725,A -85,B 0,C 180,E1 -2043.164,E2 -2043.164} C_VEL
LIN {X 0,Y 573.087,Z 573.664,A -85,B 0,C 180,E1 -2044.388,E2 -2044.388} C_VEL
LIN {X 0,Y 573.029,Z 578.872,A -85,B 0,C 180,E1 -2045.356,E2 -2045.356} C_VEL
LIN {X 0,Y 573.032,Z 583.955,A -85,B 0,C 180,E1 -2046.51,E2 -2046.51} C_VEL
LIN {X 0,Y 572.966,Z 587.926,A -85,B 0,C 180,E1 -2047.652,E2 -2047.652} C_VEL
LIN {X 0,Y 572.979,Z 590.903,A -85,B 0,C 180,E1 -2048.778,E2 -2048.778} C_VEL
LIN {X 0,Y 572.948,Z 592.966,A -85,B 0,C 180,E1 -2049.913,E2 -2049.913} C_VEL
LIN {X 0,Y 572.944,Z 594.361,A -85,B 0,C 180,E1 -2051.403,E2 -2051.403} C_VEL
LIN {X 0,Y 572.933,Z 594.247,A -85,B 0,C 180,E1 -2052.879,E2 -2052.879} C_VEL
LIN {X 0,Y 572.931,Z 592.703,A -85,B 0,C 180,E1 -2054.344,E2 -2054.344} C_VEL
LIN {X 0,Y 572.973,Z 589.713,A -85,B 0,C 180,E1 -2055.8,E2 -2055.8} C_VEL
LIN {X 0,Y 573.004,Z 585.231,A -85,B 0,C 180,E1 -2057.246,E2 -2057.246} C_VEL
LIN {X 0,Y 573.025,Z 580.788,A -85,B 0,C 180,E1 -2058.325,E2 -2058.325} C_VEL
LIN {X 0,Y 573.057,Z 574.366,A -85,B 0,C 180,E1 -2059.579,E2 -2059.579} C_VEL
LIN {X 0,Y 573.163,Z 566.403,A -85,B 0,C 180,E1 -2060.828,E2 -2060.828} C_VEL
LIN {X 0,Y 573.276,Z 558.116,A -85,B 0,C 180,E1 -2061.896,E2 -2061.896} C_VEL
LIN {X 0,Y 573.401,Z 548.193,A -85,B 0,C 180,E1 -2062.96,E2 -2062.96} C_VEL
LIN {X 0,Y 573.535,Z 537.214,A -85,B 0,C 180,E1 -2063.934,E2 -2063.934} C_VEL
LIN {X 0,Y 573.675,Z 525,A -85,B 0,C 180,E1 -2064.817,E2 -2064.817} C_VEL
LIN {X 0,Y 573.811,Z 512.991,A -85,B 0,C 180,E1 -2065.522,E2 -2065.522} C_VEL
LIN {X 0,Y 573.998,Z 499.712,A -85,B 0,C 180,E1 -2066.139,E2 -2066.139} C_VEL
LIN {X 0,Y 574.133,Z 485.172,A -85,B 0,C 180,E1 -2066.645,E2 -2066.645} C_VEL
LIN {X 0,Y 574.259,Z 471.402,A -85,B 0,C 180,E1 -2066.975,E2 -2066.975} C_VEL
LIN {X 0,Y 574.34,Z 447.799,A -85,B 0,C 180,E1 -2067.305,E2 -2067.305} C_VEL
LIN {X 0,Y 574.499,Z 338.127,A -85,B 0,C 180,E1 -2068.697,E2 -2068.697} C_VEL
LIN {X 0,Y 573.502,Z 332.818,A -85,B 0,C 180,E1 -2068.816,E2 -2068.816} C_VEL
LIN {X 0,Y 573.704,Z 314.21,A -85,B 0,C 180,E1 -2071.756,E2 -2071.756} C_VEL
LIN {X 0,Y 573.455,Z 308.779,A -85,B 0,C 180,E1 -2072.635,E2 -2072.635} C_VEL
LIN {X 0,Y 573.299,Z 307.7,A -85,B 0,C 180,E1 -2072.855,E2 -2072.855} C_VEL
LIN {X 0,Y 573.279,Z 307.702,A -85,B 0,C 180,E1 -2075.629,E2 -2075.629} C_VEL
LIN {X 0,Y 573.263,Z 307.702,A -85,B 0,C 180,E1 -2077.751,E2 -2077.751} C_VEL
LIN {X 0,Y 573.24,Z 307.701,A -85,B 0,C 180,E1 -2080.598,E2 -2080.598} C_VEL
LIN {X 0,Y 573.23,Z 307.702,A -85,B 0,C 180,E1 -2082.75,E2 -2082.75} C_VEL
LIN {X 0,Y 573.217,Z 307.707,A -85,B 0,C 180,E1 -2084.921,E2 -2084.921} C_VEL
LIN {X 0,Y 573.244,Z 307.707,A -85,B 0,C 180,E1 -2087.113,E2 -2087.113} C_VEL
LIN {X 0,Y 573.231,Z 307.7,A -85,B 0,C 180,E1 -2090.078,E2 -2090.078} C_VEL
LIN {X 0,Y 573.214,Z 307.703,A -85,B 0,C 180,E1 -2092.339,E2 -2092.339} C_VEL
LIN {X 0,Y 573.218,Z 307.706,A -85,B 0,C 180,E1 -2095.412,E2 -2095.412} C_VEL
LIN {X 0,Y 573.196,Z 307.708,A -85,B 0,C 180,E1 -2098.567,E2 -2098.567} C_VEL
LIN {X 0,Y 573.206,Z 307.713,A -85,B 0,C 180,E1 -2100.995,E2 -2100.995} C_VEL
LIN {X 0,Y 573.213,Z 307.704,A -85,B 0,C 180,E1 -2103.517,E2 -2103.517} C_VEL
LIN {X 0,Y 573.181,Z 307.707,A -85,B 0,C 180,E1 -2106.054,E2 -2106.054} C_VEL
LIN {X 0,Y 573.213,Z 307.71,A -85,B 0,C 180,E1 -2108.704,E2 -2108.704} C_VEL
LIN {X 0,Y 573.189,Z 307.707,A -85,B 0,C 180,E1 -2111.461,E2 -2111.461} C_VEL
LIN {X 0,Y 573.194,Z 307.708,A -85,B 0,C 180,E1 -2114.338,E2 -2114.338} C_VEL
LIN {X 0,Y 573.204,Z 307.705,A -85,B 0,C 180,E1 -2117.363,E2 -2117.363} C_VEL
LIN {X 0,Y 573.217,Z 307.711,A -85,B 0,C 180,E1 -2120.572,E2 -2120.572} C_VEL
LIN {X 0,Y 573.217,Z 307.705,A -85,B 0,C 180,E1 -2123.075,E2 -2123.075} C_VEL
LIN {X 0,Y 573.242,Z 307.699,A -85,B 0,C 180,E1 -2125.67,E2 -2125.67} C_VEL
LIN {X 0,Y 573.222,Z 307.706,A -85,B 0,C 180,E1 -2128.184,E2 -2128.184} C_VEL
LIN {X 0,Y 573.215,Z 307.71,A -85,B 0,C 180,E1 -2130.632,E2 -2130.632} C_VEL
LIN {X 0,Y 573.204,Z 307.703,A -85,B 0,C 180,E1 -2133.515,E2 -2133.515} C_VEL
LIN {X 0,Y 573.194,Z 307.71,A -85,B 0,C 180,E1 -2136.133,E2 -2136.133} C_VEL
LIN {X 0,Y 573.228,Z 307.701,A -85,B 0,C 180,E1 -2139.173,E2 -2139.173} C_VEL
LIN {X 0,Y 573.198,Z 307.704,A -85,B 0,C 180,E1 -2141.411,E2 -2141.411} C_VEL
LIN {X 0,Y 573.21,Z 307.711,A -85,B 0,C 180,E1 -2144.352,E2 -2144.352} C_VEL
LIN {X 0,Y 573.205,Z 307.708,A -85,B 0,C 180,E1 -2146.529,E2 -2146.529} C_VEL
LIN {X 0,Y 573.26,Z 307.697,A -85,B 0,C 180,E1 -2149.404,E2 -2149.404} C_VEL
LIN {X 0,Y 573.262,Z 307.704,A -85,B 0,C 180,E1 -2152.25,E2 -2152.25} C_VEL
LIN {X 0,Y 573.288,Z 307.693,A -85,B 0,C 180,E1 -2155.077,E2 -2155.077} C_VEL
LIN {X 0,Y 573.311,Z 307.698,A -85,B 0,C 180,E1 -2157.893,E2 -2157.893} C_VEL
LIN {X 0,Y 573.329,Z 307.689,A -85,B 0,C 180,E1 -2160.703,E2 -2160.703} C_VEL
LIN {X 0,Y 573.296,Z 307.692,A -85,B 0,C 180,E1 -2162.811,E2 -2162.811} C_VEL
LIN {X 0,Y 573.282,Z 307.699,A -85,B 0,C 180,E1 -2165.628,E2 -2165.628} C_VEL
LIN {X 0,Y 573.283,Z 307.695,A -85,B 0,C 180,E1 -2168.46,E2 -2168.46} C_VEL
LIN {X 0,Y 573.275,Z 307.697,A -85,B 0,C 180,E1 -2171.312,E2 -2171.312} C_VEL
LIN {X 0,Y 573.284,Z 307.695,A -85,B 0,C 180,E1 -2174.424,E2 -2174.424} C_VEL
LIN {X 0,Y 573.261,Z 307.698,A -85,B 0,C 180,E1 -2177.112,E2 -2177.112} C_VEL
LIN {X 0,Y 573.252,Z 307.701,A -85,B 0,C 180,E1 -2180.077,E2 -2180.077} C_VEL
LIN {X 0,Y 573.238,Z 307.702,A -85,B 0,C 180,E1 -2183.099,E2 -2183.099} C_VEL
LIN {X 0,Y 573.258,Z 307.704,A -85,B 0,C 180,E1 -2185.41,E2 -2185.41} C_VEL
LIN {X 0,Y 573.238,Z 307.699,A -85,B 0,C 180,E1 -2188.565,E2 -2188.565} C_VEL
LIN {X 0,Y 573.228,Z 307.703,A -85,B 0,C 180,E1 -2190.993,E2 -2190.993} C_VEL
LIN {X 0,Y 573.266,Z 307.704,A -85,B 0,C 180,E1 -2193.524,E2 -2193.524} C_VEL
LIN {X 0,Y 573.197,Z 307.706,A -85,B 0,C 180,E1 -2196.053,E2 -2196.053} C_VEL
LIN {X 0,Y 573.241,Z 307.7,A -85,B 0,C 180,E1 -2198.702,E2 -2198.702} C_VEL
LIN {X 0,Y 573.241,Z 307.704,A -85,B 0,C 180,E1 -2201.594,E2 -2201.594} C_VEL
LIN {X 0,Y 573.237,Z 307.699,A -85,B 0,C 180,E1 -2204.334,E2 -2204.334} C_VEL
LIN {X 0,Y 573.243,Z 307.706,A -85,B 0,C 180,E1 -2207.359,E2 -2207.359} C_VEL
LIN {X 0,Y 573.255,Z 307.699,A -85,B 0,C 180,E1 -2210.567,E2 -2210.567} C_VEL
LIN {X 0,Y 573.255,Z 307.707,A -85,B 0,C 180,E1 -2213.077,E2 -2213.077} C_VEL
LIN {X 0,Y 573.27,Z 307.697,A -85,B 0,C 180,E1 -2215.671,E2 -2215.671} C_VEL
LIN {X 0,Y 573.24,Z 307.7,A -85,B 0,C 180,E1 -2218.184,E2 -2218.184} C_VEL
LIN {X 0,Y 573.264,Z 307.702,A -85,B 0,C 180,E1 -2220.634,E2 -2220.634} C_VEL
LIN {X 0,Y 573.254,Z 307.707,A -85,B 0,C 180,E1 -2223.024,E2 -2223.024} C_VEL
LIN {X 0,Y 573.285,Z 307.813,A -85,B 0,C 180,E1 -2224.989,E2 -2224.989} C_VEL
LIN {X 0,Y 574.38,Z 313.668,A -85,B 0,C 180,E1 -2225.801,E2 -2225.801} C_VEL
LIN {X 0,Y 574.066,Z 337.178,A -85,B 0,C 180,E1 -2228.861,E2 -2228.861} C_VEL
LIN {X 0,Y 573.796,Z 360.098,A -85,B 0,C 180,E1 -2231.8,E2 -2231.8} C_VEL
LIN {X 0,Y 573.661,Z 371.415,A -85,B 0,C 180,E1 -2233.233,E2 -2233.233} C_VEL
LIN {X 0,Y 574.587,Z 377.389,A -85,B 0,C 180,E1 -2233.341,E2 -2233.341} C_VEL
LIN {X 0,Y 574.305,Z 509.858,A -85,B 0,C 180,E1 -2235.04,E2 -2235.04} C_VEL
LIN {X 0,Y 574.144,Z 524.475,A -85,B 0,C 180,E1 -2235.379,E2 -2235.379} C_VEL
LIN {X 0,Y 574.017,Z 538.826,A -85,B 0,C 180,E1 -2235.87,E2 -2235.87} C_VEL
LIN {X 0,Y 573.87,Z 551.633,A -85,B 0,C 180,E1 -2236.454,E2 -2236.454} C_VEL
LIN {X 0,Y 573.713,Z 564.092,A -85,B 0,C 180,E1 -2237.171,E2 -2237.171} C_VEL
LIN {X 0,Y 573.534,Z 576.635,A -85,B 0,C 180,E1 -2238.066,E2 -2238.066} C_VEL
LIN {X 0,Y 573.437,Z 588.171,A -85,B 0,C 180,E1 -2239.083,E2 -2239.083} C_VEL
LIN {X 0,Y 573.24,Z 597.847,A -85,B 0,C 180,E1 -2240.116,E2 -2240.116} C_VEL
LIN {X 0,Y 573.202,Z 606.168,A -85,B 0,C 180,E1 -2241.183,E2 -2241.183} C_VEL
LIN {X 0,Y 573.111,Z 614.124,A -85,B 0,C 180,E1 -2242.424,E2 -2242.424} C_VEL
LIN {X 0,Y 573.013,Z 620.525,A -85,B 0,C 180,E1 -2243.662,E2 -2243.662} C_VEL
LIN {X 0,Y 573.001,Z 624.959,A -85,B 0,C 180,E1 -2244.721,E2 -2244.721} C_VEL
LIN {X 0,Y 573.028,Z 628.441,A -85,B 0,C 180,E1 -2245.779,E2 -2245.779} C_VEL
LIN {X 0,Y 572.956,Z 631.83,A -85,B 0,C 180,E1 -2247.187,E2 -2247.187} C_VEL
LIN {X 0,Y 572.941,Z 633.832,A -85,B 0,C 180,E1 -2248.594,E2 -2248.594} C_VEL
LIN {X 0,Y 572.937,Z 634.5,A -85,B 0,C 180,E1 -2249.999,E2 -2249.999} C_VEL
LIN {X 0,Y 572.941,Z 633.834,A -85,B 0,C 180,E1 -2251.405,E2 -2251.405} C_VEL
LIN {X 0,Y 572.956,Z 631.835,A -85,B 0,C 180,E1 -2252.812,E2 -2252.812} C_VEL
LIN {X 0,Y 573.028,Z 628.447,A -85,B 0,C 180,E1 -2254.219,E2 -2254.219} C_VEL
LIN {X 0,Y 573.056,Z 623.571,A -85,B 0,C 180,E1 -2255.63,E2 -2255.63} C_VEL
LIN {X 0,Y 573.064,Z 618.823,A -85,B 0,C 180,E1 -2256.699,E2 -2256.699} C_VEL
LIN {X 0,Y 573.125,Z 612.042,A -85,B 0,C 180,E1 -2257.929,E2 -2257.929} C_VEL
LIN {X 0,Y 573.226,Z 603.564,A -85,B 0,C 180,E1 -2259.171,E2 -2259.171} C_VEL
LIN {X 0,Y 573.304,Z 594.714,A -85,B 0,C 180,E1 -2260.238,E2 -2260.238} C_VEL
LIN {X 0,Y 573.461,Z 583.998,A -85,B 0,C 180,E1 -2261.307,E2 -2261.307} C_VEL
LIN {X 0,Y 573.616,Z 573.151,A -85,B 0,C 180,E1 -2262.201,E2 -2262.201} C_VEL
LIN {X 0,Y 573.74,Z 561.269,A -85,B 0,C 180,E1 -2263.007,E2 -2263.007} C_VEL
LIN {X 0,Y 573.945,Z 548.111,A -85,B 0,C 180,E1 -2263.723,E2 -2263.723} C_VEL
LIN {X 0,Y 574.085,Z 534.837,A -85,B 0,C 180,E1 -2264.284,E2 -2264.284} C_VEL
LIN {X 0,Y 574.204,Z 520.771,A -85,B 0,C 180,E1 -2264.721,E2 -2264.721} C_VEL
LIN {X 0,Y 574.3,Z 507.182,A -85,B 0,C 180,E1 -2265.004,E2 -2265.004} C_VEL
LIN {X 0,Y 574.533,Z 376.387,A -85,B 0,C 180,E1 -2266.673,E2 -2266.673} C_VEL
LIN {X 0,Y 573.654,Z 371.337,A -85,B 0,C 180,E1 -2266.777,E2 -2266.777} C_VEL
LIN {X 0,Y 573.886,Z 350.359,A -85,B 0,C 180,E1 -2269.444,E2 -2269.444} C_VEL
LIN {X 0,Y 574.141,Z 329.697,A -85,B 0,C 180,E1 -2272.11,E2 -2272.11} C_VEL
LIN {X 0,Y 574.376,Z 313.658,A -85,B 0,C 180,E1 -2274.198,E2 -2274.198} C_VEL
LIN {X 0,Y 573.273,Z 307.704,A -85,B 0,C 180,E1 -2275.029,E2 -2275.029} C_VEL
LIN {X 0,Y 573.248,Z 307.7,A -85,B 0,C 180,E1 -2278.028,E2 -2278.028} C_VEL
LIN {X 0,Y 573.236,Z 307.709,A -85,B 0,C 180,E1 -2280.883,E2 -2280.883} C_VEL
LIN {X 0,Y 573.26,Z 307.698,A -85,B 0,C 180,E1 -2283.523,E2 -2283.523} C_VEL
LIN {X 0,Y 573.258,Z 307.697,A -85,B 0,C 180,E1 -2286.047,E2 -2286.047} C_VEL
LIN {X 0,Y 573.246,Z 307.707,A -85,B 0,C 180,E1 -2288.7,E2 -2288.7} C_VEL
LIN {X 0,Y 573.239,Z 307.699,A -85,B 0,C 180,E1 -2291.594,E2 -2291.594} C_VEL
LIN {X 0,Y 573.231,Z 307.705,A -85,B 0,C 180,E1 -2294.333,E2 -2294.333} C_VEL
LIN {X 0,Y 573.239,Z 307.7,A -85,B 0,C 180,E1 -2297.357,E2 -2297.357} C_VEL
LIN {X 0,Y 573.242,Z 307.705,A -85,B 0,C 180,E1 -2300.392,E2 -2300.392} C_VEL
LIN {X 0,Y 573.25,Z 307.7,A -85,B 0,C 180,E1 -2303.077,E2 -2303.077} C_VEL
LIN {X 0,Y 573.262,Z 307.697,A -85,B 0,C 180,E1 -2305.671,E2 -2305.671} C_VEL
LIN {X 0,Y 573.237,Z 307.706,A -85,B 0,C 180,E1 -2308.184,E2 -2308.184} C_VEL
